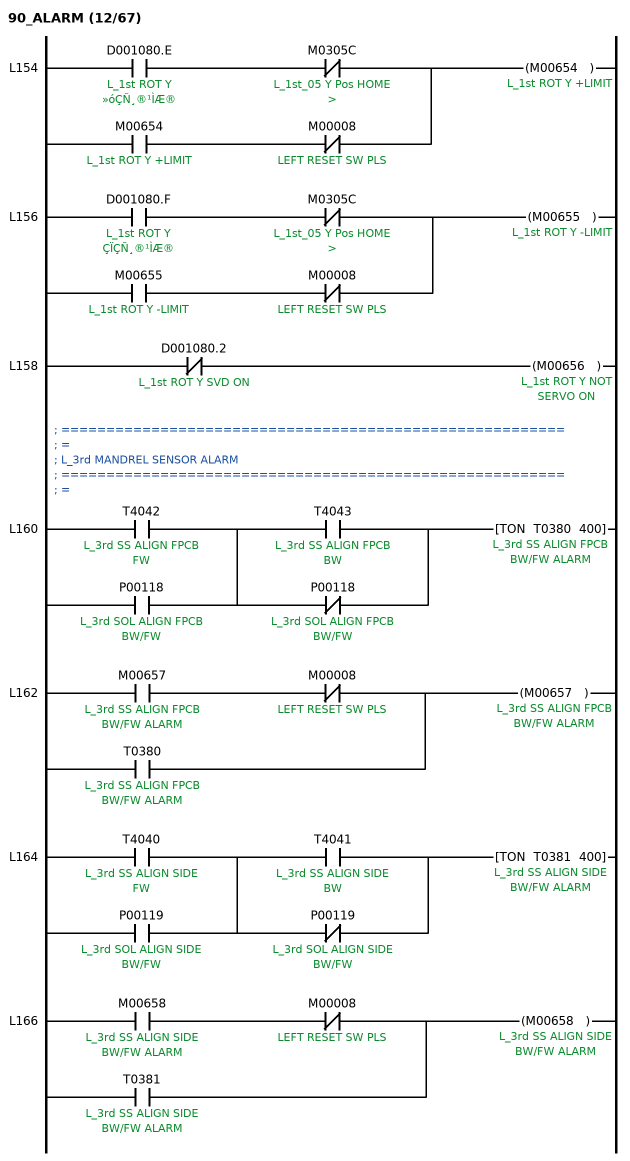
[picture p408: 90_ALARM rungs L154-L166]
; L154
LOAD      D001080.E	// L_1st ROT Y »óÇÑ¸®¹ÌÆ®
AND NOT   M0305C	// L_1st_05 Y Pos HOME >
LOAD      M00654	// L_1st ROT Y +LIMIT
AND NOT   M00008	// LEFT RESET SW PLS
OR LOAD
OUT       M00654	// L_1st ROT Y +LIMIT
; L156
LOAD      D001080.F	// L_1st ROT Y ÇÏÇÑ¸®¹ÌÆ®
AND NOT   M0305C	// L_1st_05 Y Pos HOME >
LOAD      M00655	// L_1st ROT Y -LIMIT
AND NOT   M00008	// LEFT RESET SW PLS
OR LOAD
OUT       M00655	// L_1st ROT Y -LIMIT
; L158
LOAD NOT  D001080.2	// L_1st ROT Y SVD ON
OUT       M00656	// L_1st ROT Y NOT SERVO ON
// =========================================================
// 
//        L_3rd MANDREL SENSOR ALARM
// 
// =========================================================
; L160
LOAD      T4042	// L_3rd SS ALIGN FPCB FW
OR        P00118	// L_3rd SOL ALIGN FPCB BW/FW
LOAD      T4043	// L_3rd SS ALIGN FPCB BW
OR NOT    P00118	// L_3rd SOL ALIGN FPCB BW/FW
AND LOAD
TON       T0380 400	// L_3rd SS ALIGN FPCB BW/FW ALARM
; L162
LOAD      M00657	// L_3rd SS ALIGN FPCB BW/FW ALARM
AND NOT   M00008	// LEFT RESET SW PLS
OR        T0380	// L_3rd SS ALIGN FPCB BW/FW ALARM
OUT       M00657	// L_3rd SS ALIGN FPCB BW/FW ALARM
; L164
LOAD      T4040	// L_3rd SS ALIGN SIDE FW
OR        P00119	// L_3rd SOL ALIGN SIDE BW/FW
LOAD      T4041	// L_3rd SS ALIGN SIDE BW
OR NOT    P00119	// L_3rd SOL ALIGN SIDE BW/FW
AND LOAD
TON       T0381 400	// L_3rd SS ALIGN SIDE BW/FW ALARM
; L166
LOAD      M00658	// L_3rd SS ALIGN SIDE BW/FW ALARM
AND NOT   M00008	// LEFT RESET SW PLS
OR        T0381	// L_3rd SS ALIGN SIDE BW/FW ALARM
OUT       M00658	// L_3rd SS ALIGN SIDE BW/FW ALARM

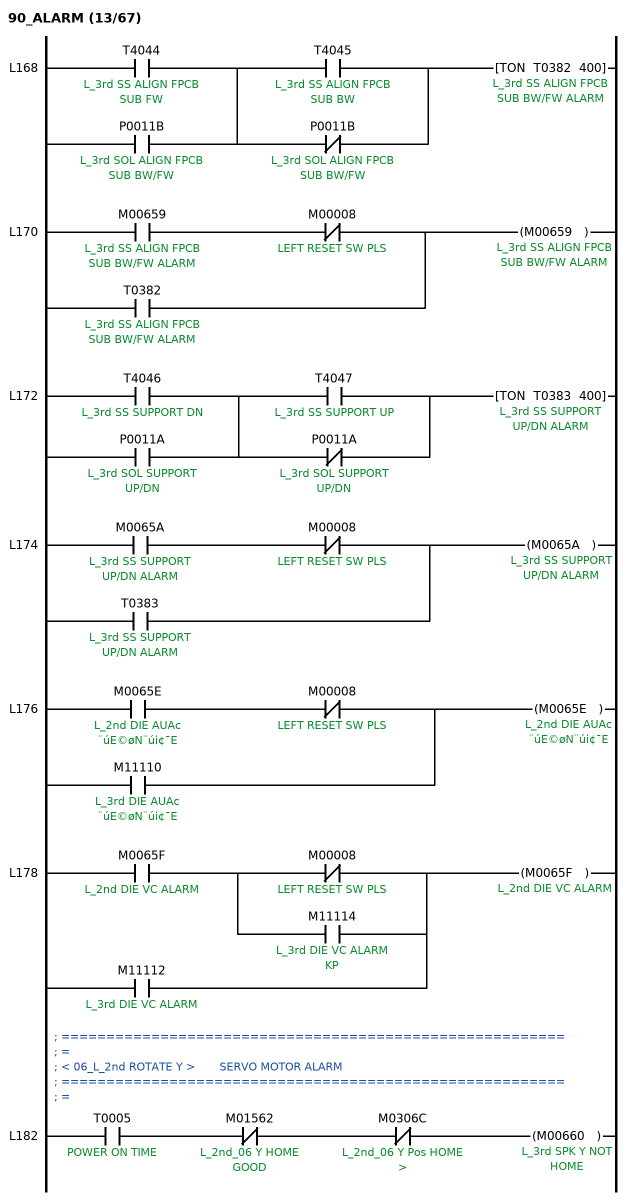
; L168
LOAD      T4044	// L_3rd SS ALIGN FPCB SUB FW
OR        P0011B	// L_3rd SOL ALIGN FPCB SUB BW/FW
LOAD      T4045	// L_3rd SS ALIGN FPCB SUB BW
OR NOT    P0011B	// L_3rd SOL ALIGN FPCB SUB BW/FW
AND LOAD
TON       T0382 400	// L_3rd SS ALIGN FPCB SUB BW/FW ALARM
; L170
LOAD      M00659	// L_3rd SS ALIGN FPCB SUB BW/FW ALARM
AND NOT   M00008	// LEFT RESET SW PLS
OR        T0382	// L_3rd SS ALIGN FPCB SUB BW/FW ALARM
OUT       M00659	// L_3rd SS ALIGN FPCB SUB BW/FW ALARM
; L172
LOAD      T4046	// L_3rd SS SUPPORT DN
OR        P0011A	// L_3rd SOL SUPPORT UP/DN
LOAD      T4047	// L_3rd SS SUPPORT UP
OR NOT    P0011A	// L_3rd SOL SUPPORT UP/DN
AND LOAD
TON       T0383 400	// L_3rd SS SUPPORT UP/DN ALARM
; L174
LOAD      M0065A	// L_3rd SS SUPPORT UP/DN ALARM
AND NOT   M00008	// LEFT RESET SW PLS
OR        T0383	// L_3rd SS SUPPORT UP/DN ALARM
OUT       M0065A	// L_3rd SS SUPPORT UP/DN ALARM
; L176
LOAD      M0065E	// L_2nd DIE AUAc ¨úE©øN¨úi¢¯E
AND NOT   M00008	// LEFT RESET SW PLS
OR        M11110	// L_3rd DIE AUAc ¨úE©øN¨úi¢¯E
OUT       M0065E	// L_2nd DIE AUAc ¨úE©øN¨úi¢¯E
; L178
LOAD      M0065F	// L_2nd DIE VC ALARM
LOAD NOT  M00008	// LEFT RESET SW PLS
OR        M11114	// L_3rd DIE VC ALARM KP
AND LOAD
OR        M11112	// L_3rd DIE VC ALARM
OUT       M0065F	// L_2nd DIE VC ALARM
// =========================================================
// 
//        < 06_L_2nd ROTATE Y >       SERVO MOTOR ALARM
// 
// =========================================================
; L182
LOAD      T0005	// POWER ON TIME
AND NOT   M01562	// L_2nd_06 Y HOME GOOD
AND NOT   M0306C	// L_2nd_06 Y Pos HOME >
OUT       M00660	// L_3rd SPK Y NOT HOME

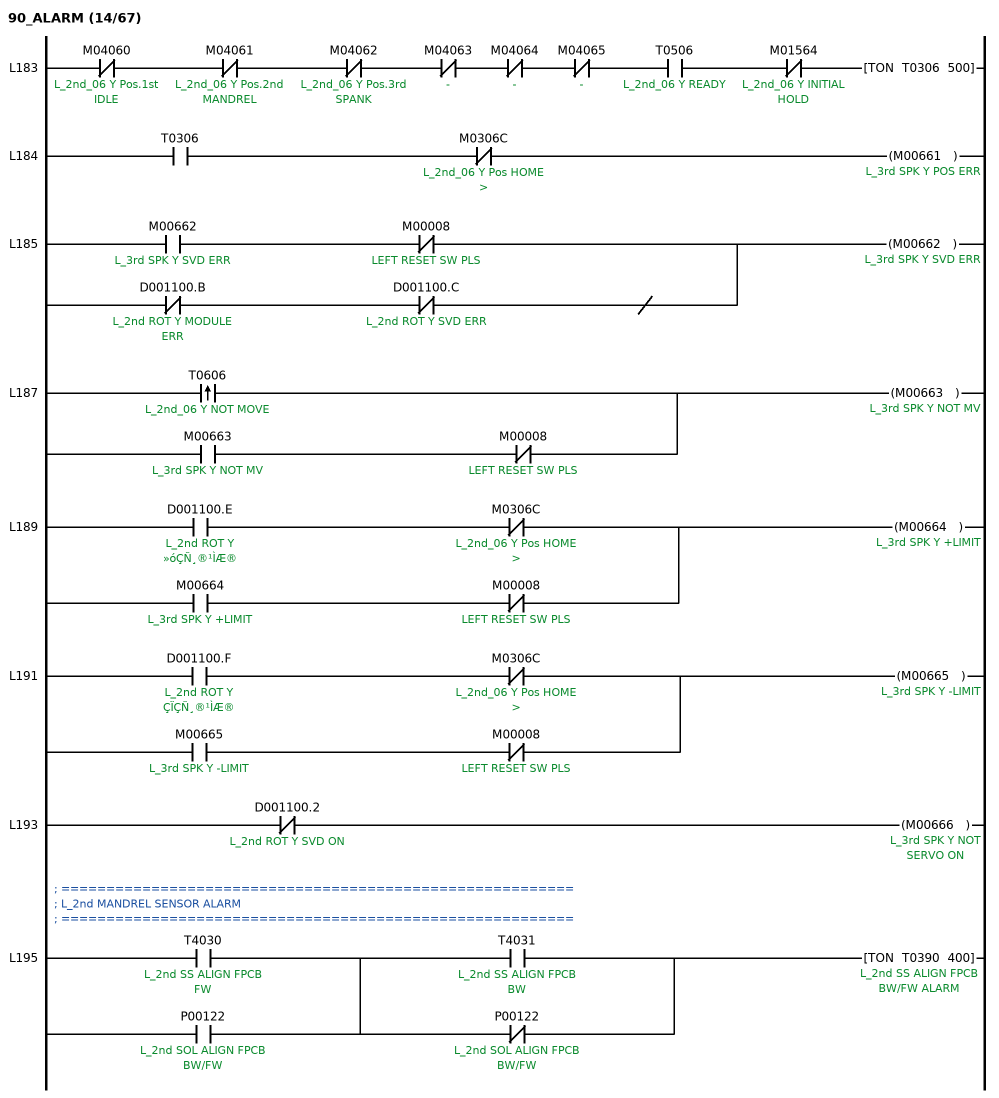
; L183
LOAD NOT  M04060	// L_2nd_06 Y Pos.1st IDLE
AND NOT   M04061	// L_2nd_06 Y Pos.2nd MANDREL
AND NOT   M04062	// L_2nd_06 Y Pos.3rd SPANK
AND NOT   M04063	// -
AND NOT   M04064	// -
AND NOT   M04065	// -
AND       T0506	// L_2nd_06 Y READY
AND NOT   M01564	// L_2nd_06 Y INITIAL HOLD
TON       T0306 500
; L184
LOAD      T0306
AND NOT   M0306C	// L_2nd_06 Y Pos HOME >
OUT       M00661	// L_3rd SPK Y POS ERR
; L185
LOAD      M00662	// L_3rd SPK Y SVD ERR
AND NOT   M00008	// LEFT RESET SW PLS
LOAD NOT  D001100.B	// L_2nd ROT Y MODULE ERR
AND NOT   D001100.C	// L_2nd ROT Y SVD ERR
NOT
OR LOAD
OUT       M00662	// L_3rd SPK Y SVD ERR
; L187
LOADP     T0606	// L_2nd_06 Y NOT MOVE
LOAD      M00663	// L_3rd SPK Y NOT MV
AND NOT   M00008	// LEFT RESET SW PLS
OR LOAD
OUT       M00663	// L_3rd SPK Y NOT MV
; L189
LOAD      D001100.E	// L_2nd ROT Y »óÇÑ¸®¹ÌÆ®
AND NOT   M0306C	// L_2nd_06 Y Pos HOME >
LOAD      M00664	// L_3rd SPK Y +LIMIT
AND NOT   M00008	// LEFT RESET SW PLS
OR LOAD
OUT       M00664	// L_3rd SPK Y +LIMIT
; L191
LOAD      D001100.F	// L_2nd ROT Y ÇÏÇÑ¸®¹ÌÆ®
AND NOT   M0306C	// L_2nd_06 Y Pos HOME >
LOAD      M00665	// L_3rd SPK Y -LIMIT
AND NOT   M00008	// LEFT RESET SW PLS
OR LOAD
OUT       M00665	// L_3rd SPK Y -LIMIT
; L193
LOAD NOT  D001100.2	// L_2nd ROT Y SVD ON
OUT       M00666	// L_3rd SPK Y NOT SERVO ON
// =========================================================
// 
//        L_2nd MANDREL SENSOR ALARM
// 
// =========================================================
; L195
LOAD      T4030	// L_2nd SS ALIGN FPCB FW
OR        P00122	// L_2nd SOL ALIGN FPCB BW/FW
LOAD      T4031	// L_2nd SS ALIGN FPCB BW
OR NOT    P00122	// L_2nd SOL ALIGN FPCB BW/FW
AND LOAD
TON       T0390 400	// L_2nd SS ALIGN FPCB BW/FW ALARM

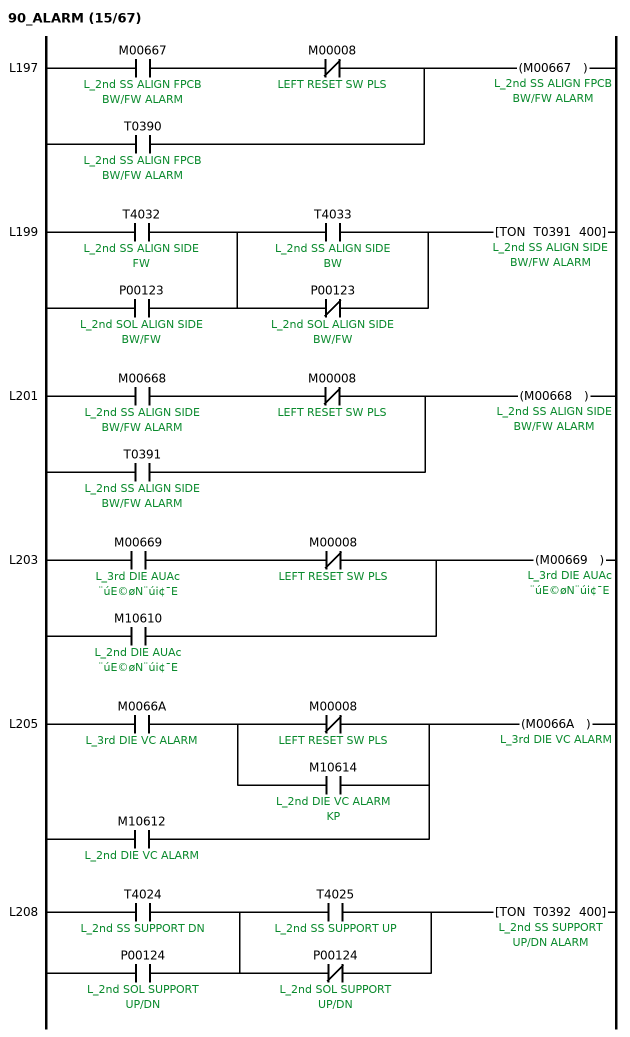
; L197
LOAD      M00667	// L_2nd SS ALIGN FPCB BW/FW ALARM
AND NOT   M00008	// LEFT RESET SW PLS
OR        T0390	// L_2nd SS ALIGN FPCB BW/FW ALARM
OUT       M00667	// L_2nd SS ALIGN FPCB BW/FW ALARM
; L199
LOAD      T4032	// L_2nd SS ALIGN SIDE FW
OR        P00123	// L_2nd SOL ALIGN SIDE BW/FW
LOAD      T4033	// L_2nd SS ALIGN SIDE BW
OR NOT    P00123	// L_2nd SOL ALIGN SIDE BW/FW
AND LOAD
TON       T0391 400	// L_2nd SS ALIGN SIDE BW/FW ALARM
; L201
LOAD      M00668	// L_2nd SS ALIGN SIDE BW/FW ALARM
AND NOT   M00008	// LEFT RESET SW PLS
OR        T0391	// L_2nd SS ALIGN SIDE BW/FW ALARM
OUT       M00668	// L_2nd SS ALIGN SIDE BW/FW ALARM
; L203
LOAD      M00669	// L_3rd DIE AUAc ¨úE©øN¨úi¢¯E
AND NOT   M00008	// LEFT RESET SW PLS
OR        M10610	// L_2nd DIE AUAc ¨úE©øN¨úi¢¯E
OUT       M00669	// L_3rd DIE AUAc ¨úE©øN¨úi¢¯E
; L205
LOAD      M0066A	// L_3rd DIE VC ALARM
LOAD NOT  M00008	// LEFT RESET SW PLS
OR        M10614	// L_2nd DIE VC ALARM KP
AND LOAD
OR        M10612	// L_2nd DIE VC ALARM
OUT       M0066A	// L_3rd DIE VC ALARM
; L208
LOAD      T4024	// L_2nd SS SUPPORT DN
OR        P00124	// L_2nd SOL SUPPORT UP/DN
LOAD      T4025	// L_2nd SS SUPPORT UP
OR NOT    P00124	// L_2nd SOL SUPPORT UP/DN
AND LOAD
TON       T0392 400	// L_2nd SS SUPPORT UP/DN ALARM

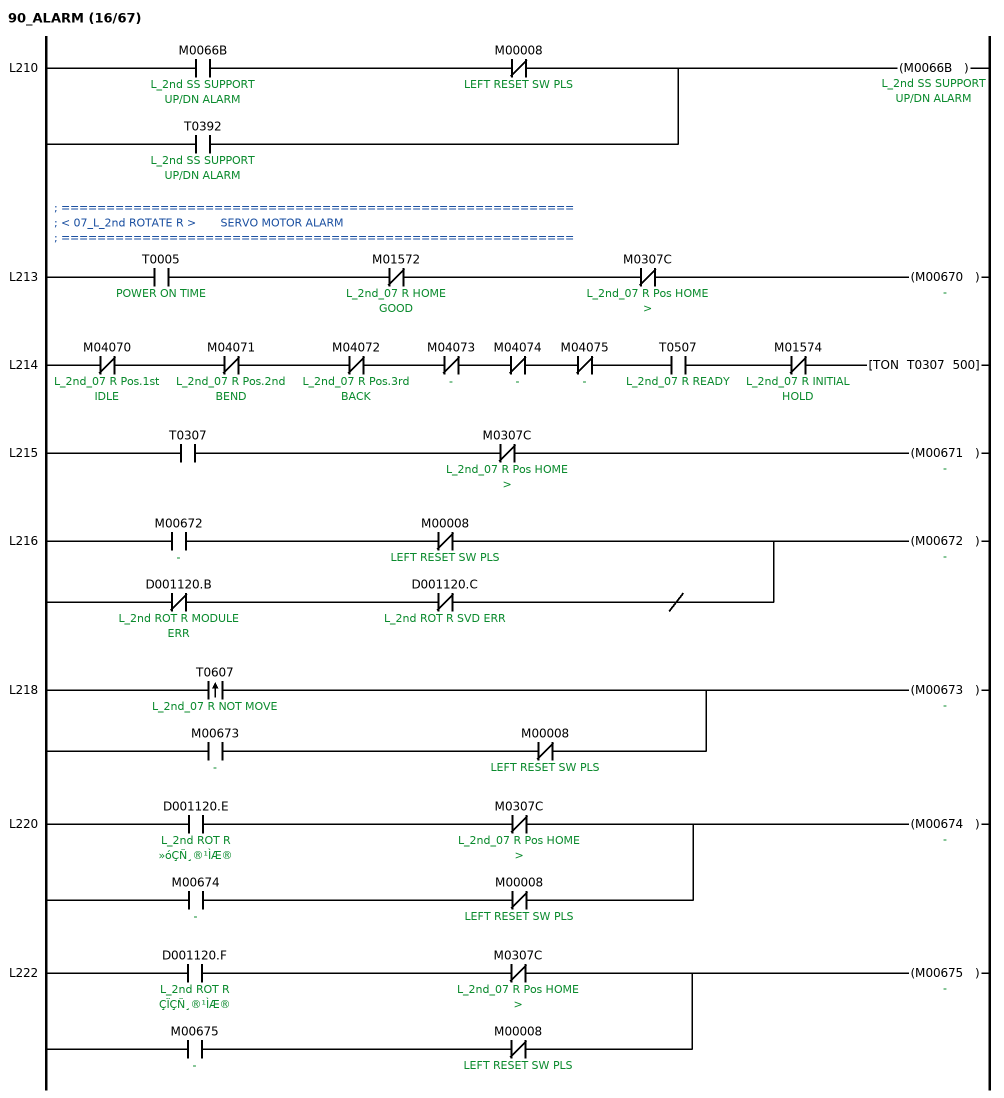
; L210
LOAD      M0066B	// L_2nd SS SUPPORT UP/DN ALARM
AND NOT   M00008	// LEFT RESET SW PLS
OR        T0392	// L_2nd SS SUPPORT UP/DN ALARM
OUT       M0066B	// L_2nd SS SUPPORT UP/DN ALARM
// =========================================================
// 
//        < 07_L_2nd ROTATE R >       SERVO MOTOR ALARM
// 
// =========================================================
; L213
LOAD      T0005	// POWER ON TIME
AND NOT   M01572	// L_2nd_07 R HOME GOOD
AND NOT   M0307C	// L_2nd_07 R Pos HOME >
OUT       M00670	// -
; L214
LOAD NOT  M04070	// L_2nd_07 R Pos.1st IDLE
AND NOT   M04071	// L_2nd_07 R Pos.2nd BEND
AND NOT   M04072	// L_2nd_07 R Pos.3rd BACK
AND NOT   M04073	// -
AND NOT   M04074	// -
AND NOT   M04075	// -
AND       T0507	// L_2nd_07 R READY
AND NOT   M01574	// L_2nd_07 R INITIAL HOLD
TON       T0307 500
; L215
LOAD      T0307
AND NOT   M0307C	// L_2nd_07 R Pos HOME >
OUT       M00671	// -
; L216
LOAD      M00672	// -
AND NOT   M00008	// LEFT RESET SW PLS
LOAD NOT  D001120.B	// L_2nd ROT R MODULE ERR
AND NOT   D001120.C	// L_2nd ROT R SVD ERR
NOT
OR LOAD
OUT       M00672	// -
; L218
LOADP     T0607	// L_2nd_07 R NOT MOVE
LOAD      M00673	// -
AND NOT   M00008	// LEFT RESET SW PLS
OR LOAD
OUT       M00673	// -
; L220
LOAD      D001120.E	// L_2nd ROT R »óÇÑ¸®¹ÌÆ®
AND NOT   M0307C	// L_2nd_07 R Pos HOME >
LOAD      M00674	// -
AND NOT   M00008	// LEFT RESET SW PLS
OR LOAD
OUT       M00674	// -
; L222
LOAD      D001120.F	// L_2nd ROT R ÇÏÇÑ¸®¹ÌÆ®
AND NOT   M0307C	// L_2nd_07 R Pos HOME >
LOAD      M00675	// -
AND NOT   M00008	// LEFT RESET SW PLS
OR LOAD
OUT       M00675	// -

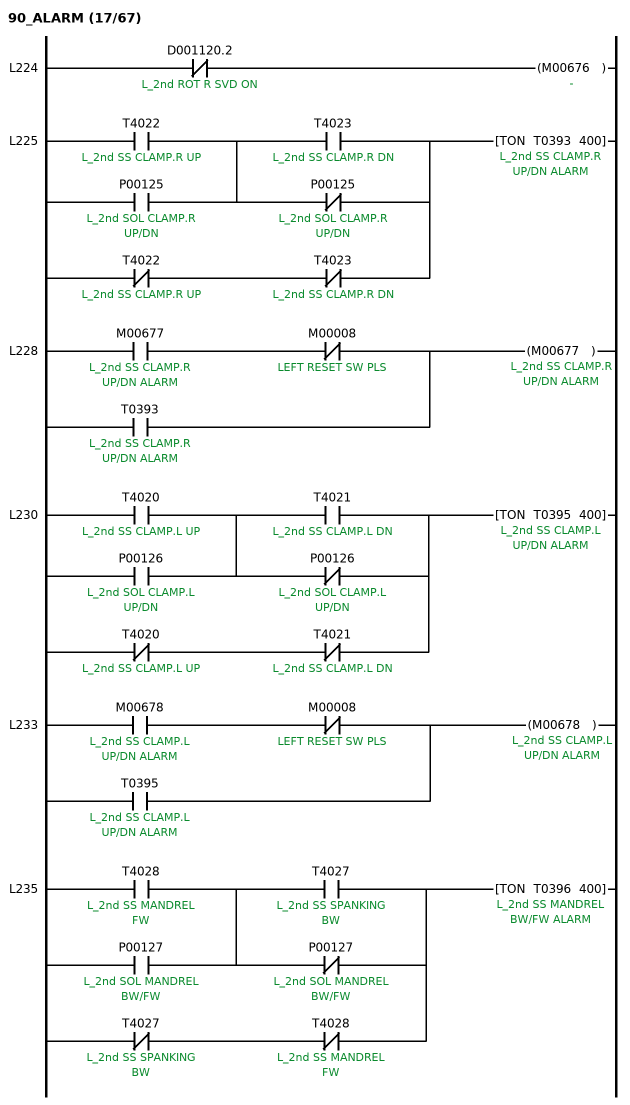
; L224
LOAD NOT  D001120.2	// L_2nd ROT R SVD ON
OUT       M00676	// -
; L225
LOAD      T4022	// L_2nd SS CLAMP.R UP
OR        P00125	// L_2nd SOL CLAMP.R UP/DN
LOAD      T4023	// L_2nd SS CLAMP.R DN
OR NOT    P00125	// L_2nd SOL CLAMP.R UP/DN
AND LOAD
LOAD NOT  T4022	// L_2nd SS CLAMP.R UP
AND NOT   T4023	// L_2nd SS CLAMP.R DN
OR LOAD
TON       T0393 400	// L_2nd SS CLAMP.R UP/DN ALARM
; L228
LOAD      M00677	// L_2nd SS CLAMP.R UP/DN ALARM
AND NOT   M00008	// LEFT RESET SW PLS
OR        T0393	// L_2nd SS CLAMP.R UP/DN ALARM
OUT       M00677	// L_2nd SS CLAMP.R UP/DN ALARM
; L230
LOAD      T4020	// L_2nd SS CLAMP.L UP
OR        P00126	// L_2nd SOL CLAMP.L UP/DN
LOAD      T4021	// L_2nd SS CLAMP.L DN
OR NOT    P00126	// L_2nd SOL CLAMP.L UP/DN
AND LOAD
LOAD NOT  T4020	// L_2nd SS CLAMP.L UP
AND NOT   T4021	// L_2nd SS CLAMP.L DN
OR LOAD
TON       T0395 400	// L_2nd SS CLAMP.L UP/DN ALARM
; L233
LOAD      M00678	// L_2nd SS CLAMP.L UP/DN ALARM
AND NOT   M00008	// LEFT RESET SW PLS
OR        T0395	// L_2nd SS CLAMP.L UP/DN ALARM
OUT       M00678	// L_2nd SS CLAMP.L UP/DN ALARM
; L235
LOAD      T4028	// L_2nd SS MANDREL FW
OR        P00127	// L_2nd SOL MANDREL BW/FW
LOAD      T4027	// L_2nd SS SPANKING BW
OR NOT    P00127	// L_2nd SOL MANDREL BW/FW
AND LOAD
LOAD NOT  T4027	// L_2nd SS SPANKING BW
AND NOT   T4028	// L_2nd SS MANDREL FW
OR LOAD
TON       T0396 400	// L_2nd SS MANDREL BW/FW ALARM

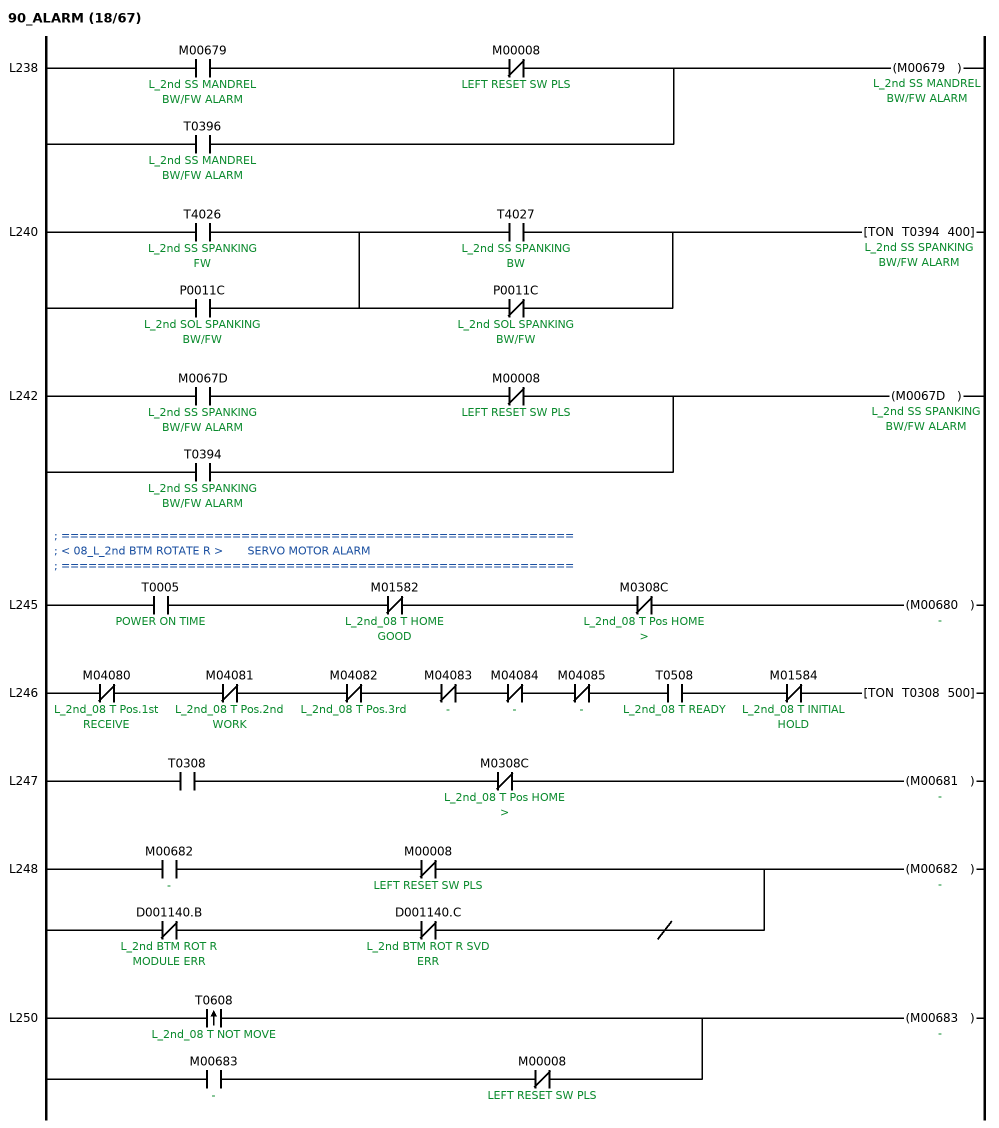
; L238
LOAD      M00679	// L_2nd SS MANDREL BW/FW ALARM
AND NOT   M00008	// LEFT RESET SW PLS
OR        T0396	// L_2nd SS MANDREL BW/FW ALARM
OUT       M00679	// L_2nd SS MANDREL BW/FW ALARM
; L240
LOAD      T4026	// L_2nd SS SPANKING FW
OR        P0011C	// L_2nd SOL SPANKING BW/FW
LOAD      T4027	// L_2nd SS SPANKING BW
OR NOT    P0011C	// L_2nd SOL SPANKING BW/FW
AND LOAD
TON       T0394 400	// L_2nd SS SPANKING BW/FW ALARM
; L242
LOAD      M0067D	// L_2nd SS SPANKING BW/FW ALARM
AND NOT   M00008	// LEFT RESET SW PLS
OR        T0394	// L_2nd SS SPANKING BW/FW ALARM
OUT       M0067D	// L_2nd SS SPANKING BW/FW ALARM
// =========================================================
// 
//        < 08_L_2nd BTM ROTATE R >       SERVO MOTOR ALARM
// 
// =========================================================
; L245
LOAD      T0005	// POWER ON TIME
AND NOT   M01582	// L_2nd_08 T HOME GOOD
AND NOT   M0308C	// L_2nd_08 T Pos HOME >
OUT       M00680	// -
; L246
LOAD NOT  M04080	// L_2nd_08 T Pos.1st RECEIVE
AND NOT   M04081	// L_2nd_08 T Pos.2nd WORK
AND NOT   M04082	// L_2nd_08 T Pos.3rd
AND NOT   M04083	// -
AND NOT   M04084	// -
AND NOT   M04085	// -
AND       T0508	// L_2nd_08 T READY
AND NOT   M01584	// L_2nd_08 T INITIAL HOLD
TON       T0308 500
; L247
LOAD      T0308
AND NOT   M0308C	// L_2nd_08 T Pos HOME >
OUT       M00681	// -
; L248
LOAD      M00682	// -
AND NOT   M00008	// LEFT RESET SW PLS
LOAD NOT  D001140.B	// L_2nd BTM ROT R MODULE ERR
AND NOT   D001140.C	// L_2nd BTM ROT R SVD ERR
NOT
OR LOAD
OUT       M00682	// -
; L250
LOADP     T0608	// L_2nd_08 T NOT MOVE
LOAD      M00683	// -
AND NOT   M00008	// LEFT RESET SW PLS
OR LOAD
OUT       M00683	// -

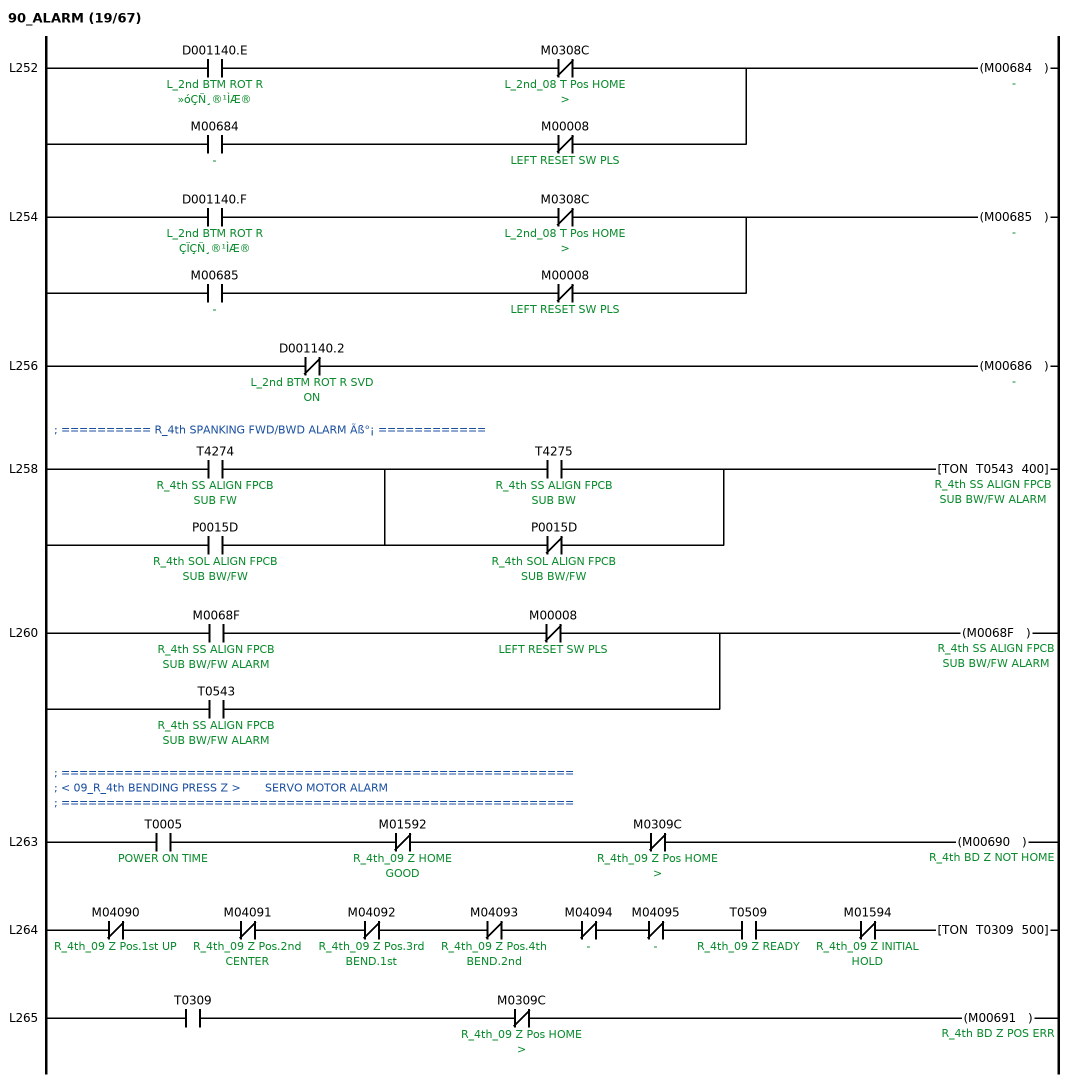
; L252
LOAD      D001140.E	// L_2nd BTM ROT R »óÇÑ¸®¹ÌÆ®
AND NOT   M0308C	// L_2nd_08 T Pos HOME >
LOAD      M00684	// -
AND NOT   M00008	// LEFT RESET SW PLS
OR LOAD
OUT       M00684	// -
; L254
LOAD      D001140.F	// L_2nd BTM ROT R ÇÏÇÑ¸®¹ÌÆ®
AND NOT   M0308C	// L_2nd_08 T Pos HOME >
LOAD      M00685	// -
AND NOT   M00008	// LEFT RESET SW PLS
OR LOAD
OUT       M00685	// -
; L256
LOAD NOT  D001140.2	// L_2nd BTM ROT R SVD ON
OUT       M00686	// -
// ========== R_4th SPANKING FWD/BWD ALARM Ãß°¡ ============
; L258
LOAD      T4274	// R_4th SS ALIGN FPCB SUB FW
OR        P0015D	// R_4th SOL ALIGN FPCB SUB BW/FW
LOAD      T4275	// R_4th SS ALIGN FPCB SUB BW
OR NOT    P0015D	// R_4th SOL ALIGN FPCB SUB BW/FW
AND LOAD
TON       T0543 400	// R_4th SS ALIGN FPCB SUB BW/FW ALARM
; L260
LOAD      M0068F	// R_4th SS ALIGN FPCB SUB BW/FW ALARM
AND NOT   M00008	// LEFT RESET SW PLS
OR        T0543	// R_4th SS ALIGN FPCB SUB BW/FW ALARM
OUT       M0068F	// R_4th SS ALIGN FPCB SUB BW/FW ALARM
// =========================================================
// 
//        < 09_R_4th BENDING PRESS Z >       SERVO MOTOR ALARM
// 
// =========================================================
; L263
LOAD      T0005	// POWER ON TIME
AND NOT   M01592	// R_4th_09 Z HOME GOOD
AND NOT   M0309C	// R_4th_09 Z Pos HOME >
OUT       M00690	// R_4th BD Z NOT HOME
; L264
LOAD NOT  M04090	// R_4th_09 Z Pos.1st UP
AND NOT   M04091	// R_4th_09 Z Pos.2nd CENTER
AND NOT   M04092	// R_4th_09 Z Pos.3rd BEND.1st
AND NOT   M04093	// R_4th_09 Z Pos.4th BEND.2nd
AND NOT   M04094	// -
AND NOT   M04095	// -
AND       T0509	// R_4th_09 Z READY
AND NOT   M01594	// R_4th_09 Z INITIAL HOLD
TON       T0309 500
; L265
LOAD      T0309
AND NOT   M0309C	// R_4th_09 Z Pos HOME >
OUT       M00691	// R_4th BD Z POS ERR

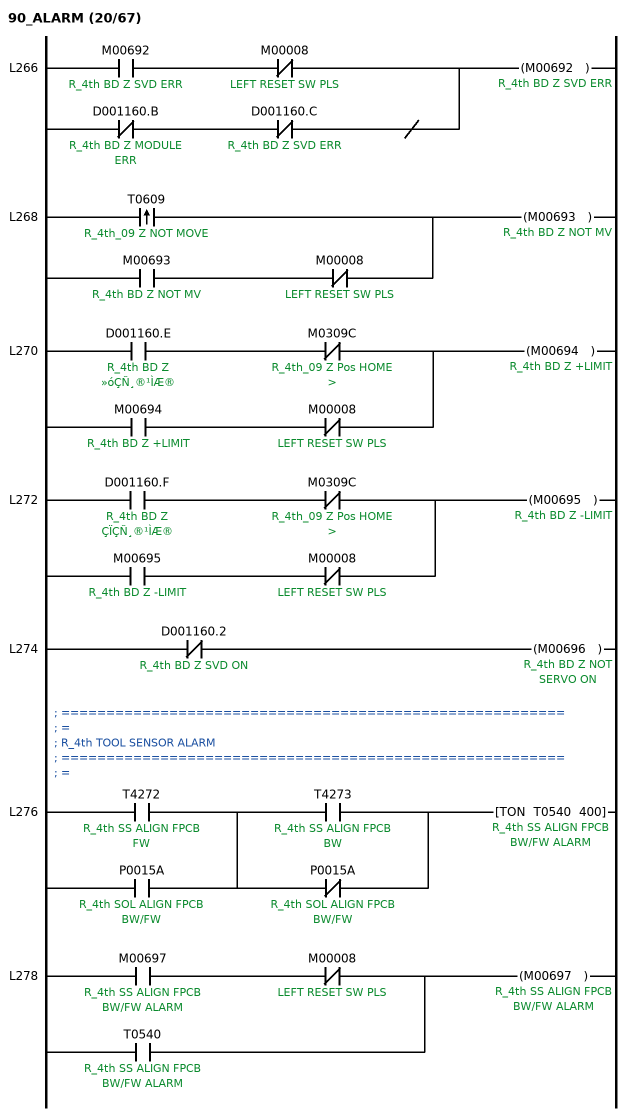
; L266
LOAD      M00692	// R_4th BD Z SVD ERR
AND NOT   M00008	// LEFT RESET SW PLS
LOAD NOT  D001160.B	// R_4th BD Z MODULE ERR
AND NOT   D001160.C	// R_4th BD Z SVD ERR
NOT
OR LOAD
OUT       M00692	// R_4th BD Z SVD ERR
; L268
LOADP     T0609	// R_4th_09 Z NOT MOVE
LOAD      M00693	// R_4th BD Z NOT MV
AND NOT   M00008	// LEFT RESET SW PLS
OR LOAD
OUT       M00693	// R_4th BD Z NOT MV
; L270
LOAD      D001160.E	// R_4th BD Z »óÇÑ¸®¹ÌÆ®
AND NOT   M0309C	// R_4th_09 Z Pos HOME >
LOAD      M00694	// R_4th BD Z +LIMIT
AND NOT   M00008	// LEFT RESET SW PLS
OR LOAD
OUT       M00694	// R_4th BD Z +LIMIT
; L272
LOAD      D001160.F	// R_4th BD Z ÇÏÇÑ¸®¹ÌÆ®
AND NOT   M0309C	// R_4th_09 Z Pos HOME >
LOAD      M00695	// R_4th BD Z -LIMIT
AND NOT   M00008	// LEFT RESET SW PLS
OR LOAD
OUT       M00695	// R_4th BD Z -LIMIT
; L274
LOAD NOT  D001160.2	// R_4th BD Z SVD ON
OUT       M00696	// R_4th BD Z NOT SERVO ON
// =========================================================
// 
//        R_4th TOOL SENSOR ALARM
// 
// =========================================================
; L276
LOAD      T4272	// R_4th SS ALIGN FPCB FW
OR        P0015A	// R_4th SOL ALIGN FPCB BW/FW
LOAD      T4273	// R_4th SS ALIGN FPCB BW
OR NOT    P0015A	// R_4th SOL ALIGN FPCB BW/FW
AND LOAD
TON       T0540 400	// R_4th SS ALIGN FPCB BW/FW ALARM
; L278
LOAD      M00697	// R_4th SS ALIGN FPCB BW/FW ALARM
AND NOT   M00008	// LEFT RESET SW PLS
OR        T0540	// R_4th SS ALIGN FPCB BW/FW ALARM
OUT       M00697	// R_4th SS ALIGN FPCB BW/FW ALARM

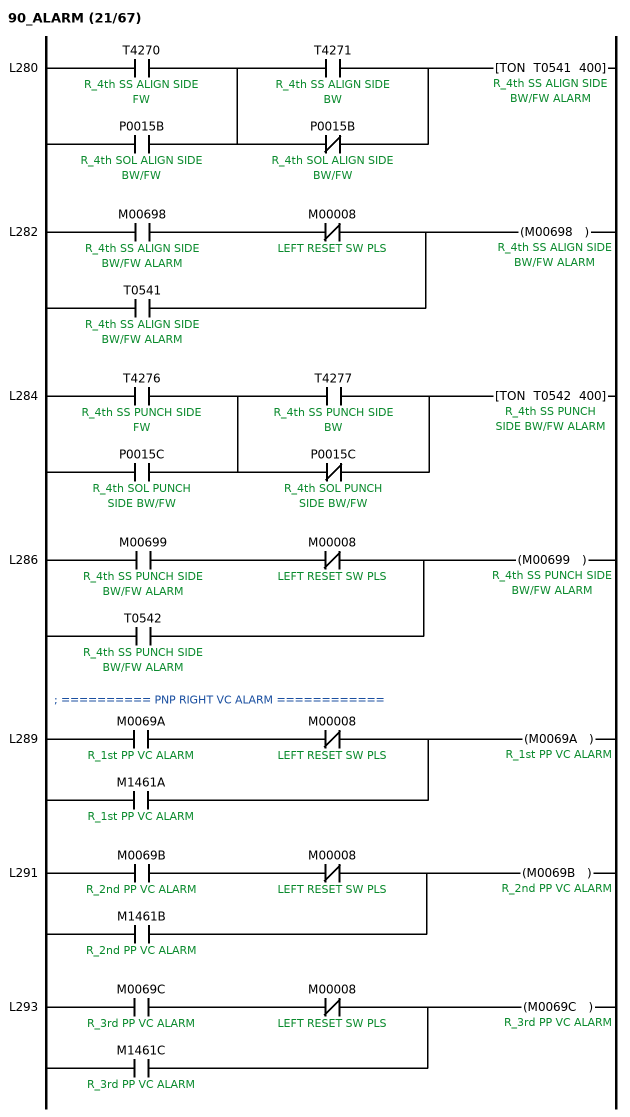
; L280
LOAD      T4270	// R_4th SS ALIGN SIDE FW
OR        P0015B	// R_4th SOL ALIGN SIDE BW/FW
LOAD      T4271	// R_4th SS ALIGN SIDE BW
OR NOT    P0015B	// R_4th SOL ALIGN SIDE BW/FW
AND LOAD
TON       T0541 400	// R_4th SS ALIGN SIDE BW/FW ALARM
; L282
LOAD      M00698	// R_4th SS ALIGN SIDE BW/FW ALARM
AND NOT   M00008	// LEFT RESET SW PLS
OR        T0541	// R_4th SS ALIGN SIDE BW/FW ALARM
OUT       M00698	// R_4th SS ALIGN SIDE BW/FW ALARM
; L284
LOAD      T4276	// R_4th SS PUNCH SIDE FW
OR        P0015C	// R_4th SOL PUNCH SIDE BW/FW
LOAD      T4277	// R_4th SS PUNCH SIDE BW
OR NOT    P0015C	// R_4th SOL PUNCH SIDE BW/FW
AND LOAD
TON       T0542 400	// R_4th SS PUNCH SIDE BW/FW ALARM
; L286
LOAD      M00699	// R_4th SS PUNCH SIDE BW/FW ALARM
AND NOT   M00008	// LEFT RESET SW PLS
OR        T0542	// R_4th SS PUNCH SIDE BW/FW ALARM
OUT       M00699	// R_4th SS PUNCH SIDE BW/FW ALARM
// ========== PNP RIGHT VC ALARM ============
; L289
LOAD      M0069A	// R_1st PP VC ALARM
AND NOT   M00008	// LEFT RESET SW PLS
OR        M1461A	// R_1st PP VC ALARM
OUT       M0069A	// R_1st PP VC ALARM
; L291
LOAD      M0069B	// R_2nd PP VC ALARM
AND NOT   M00008	// LEFT RESET SW PLS
OR        M1461B	// R_2nd PP VC ALARM
OUT       M0069B	// R_2nd PP VC ALARM
; L293
LOAD      M0069C	// R_3rd PP VC ALARM
AND NOT   M00008	// LEFT RESET SW PLS
OR        M1461C	// R_3rd PP VC ALARM
OUT       M0069C	// R_3rd PP VC ALARM

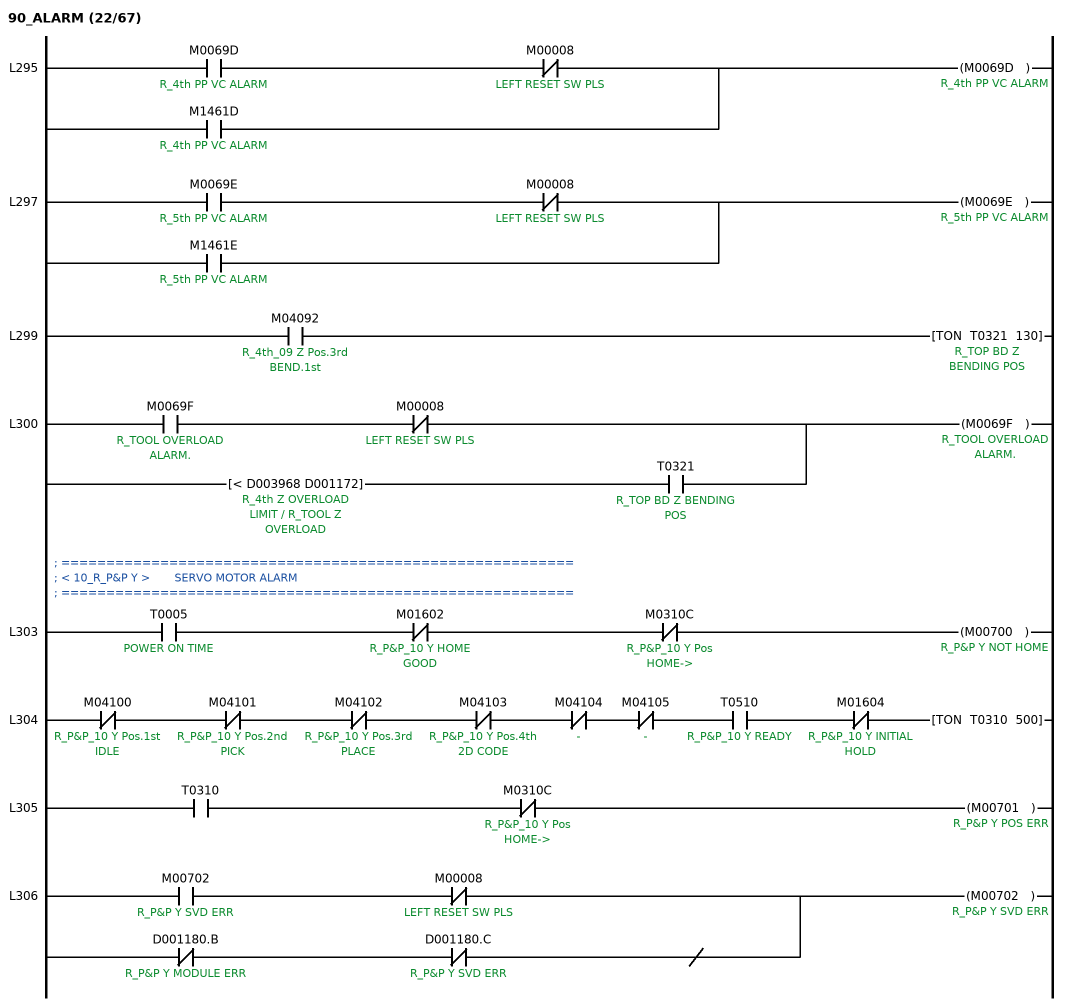
; L295
LOAD      M0069D	// R_4th PP VC ALARM
AND NOT   M00008	// LEFT RESET SW PLS
OR        M1461D	// R_4th PP VC ALARM
OUT       M0069D	// R_4th PP VC ALARM
; L297
LOAD      M0069E	// R_5th PP VC ALARM
AND NOT   M00008	// LEFT RESET SW PLS
OR        M1461E	// R_5th PP VC ALARM
OUT       M0069E	// R_5th PP VC ALARM
; L299
LOAD      M04092	// R_4th_09 Z Pos.3rd BEND.1st
TON       T0321 130	// R_TOP BD Z BENDING POS
; L300
LOAD      M0069F	// R_TOOL OVERLOAD ALARM.
AND NOT   M00008	// LEFT RESET SW PLS
LOAD<     D003968 D001172	// R_4th Z OVERLOAD LIMIT / R_TOOL Z OVERLOAD
AND       T0321	// R_TOP BD Z BENDING POS
OR LOAD
OUT       M0069F	// R_TOOL OVERLOAD ALARM.
// =========================================================
// 
//        < 10_R_P&P Y >       SERVO MOTOR ALARM
// 
// =========================================================
; L303
LOAD      T0005	// POWER ON TIME
AND NOT   M01602	// R_P&P_10 Y HOME GOOD
AND NOT   M0310C	// R_P&P_10 Y Pos HOME->
OUT       M00700	// R_P&P Y NOT HOME
; L304
LOAD NOT  M04100	// R_P&P_10 Y Pos.1st IDLE
AND NOT   M04101	// R_P&P_10 Y Pos.2nd PICK
AND NOT   M04102	// R_P&P_10 Y Pos.3rd PLACE
AND NOT   M04103	// R_P&P_10 Y Pos.4th 2D CODE
AND NOT   M04104	// -
AND NOT   M04105	// -
AND       T0510	// R_P&P_10 Y READY
AND NOT   M01604	// R_P&P_10 Y INITIAL HOLD
TON       T0310 500
; L305
LOAD      T0310
AND NOT   M0310C	// R_P&P_10 Y Pos HOME->
OUT       M00701	// R_P&P Y POS ERR
; L306
LOAD      M00702	// R_P&P Y SVD ERR
AND NOT   M00008	// LEFT RESET SW PLS
LOAD NOT  D001180.B	// R_P&P Y MODULE ERR
AND NOT   D001180.C	// R_P&P Y SVD ERR
NOT
OR LOAD
OUT       M00702	// R_P&P Y SVD ERR

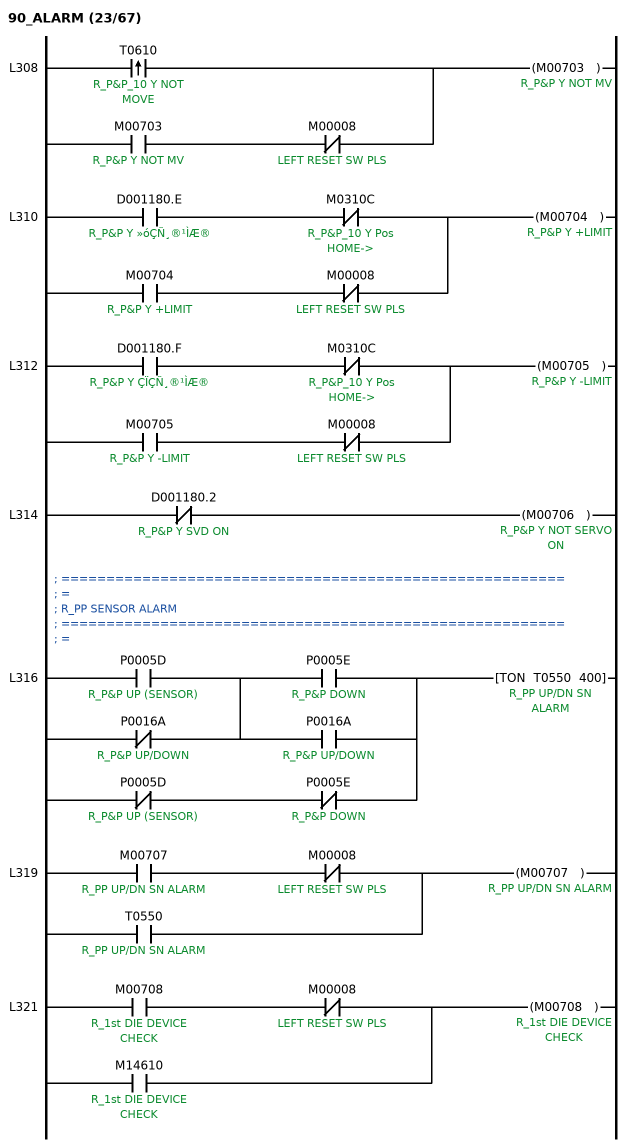
; L308
LOADP     T0610	// R_P&P_10 Y NOT MOVE
LOAD      M00703	// R_P&P Y NOT MV
AND NOT   M00008	// LEFT RESET SW PLS
OR LOAD
OUT       M00703	// R_P&P Y NOT MV
; L310
LOAD      D001180.E	// R_P&P Y »óÇÑ¸®¹ÌÆ®
AND NOT   M0310C	// R_P&P_10 Y Pos HOME->
LOAD      M00704	// R_P&P Y +LIMIT
AND NOT   M00008	// LEFT RESET SW PLS
OR LOAD
OUT       M00704	// R_P&P Y +LIMIT
; L312
LOAD      D001180.F	// R_P&P Y ÇÏÇÑ¸®¹ÌÆ®
AND NOT   M0310C	// R_P&P_10 Y Pos HOME->
LOAD      M00705	// R_P&P Y -LIMIT
AND NOT   M00008	// LEFT RESET SW PLS
OR LOAD
OUT       M00705	// R_P&P Y -LIMIT
; L314
LOAD NOT  D001180.2	// R_P&P Y SVD ON
OUT       M00706	// R_P&P Y NOT SERVO ON
// =========================================================
// 
//       R_PP SENSOR ALARM
// 
// =========================================================
; L316
LOAD      P0005D	// R_P&P UP (SENSOR)
OR NOT    P0016A	// R_P&P UP/DOWN
LOAD      P0005E	// R_P&P DOWN
OR        P0016A	// R_P&P UP/DOWN
AND LOAD
LOAD NOT  P0005D	// R_P&P UP (SENSOR)
AND NOT   P0005E	// R_P&P DOWN
OR LOAD
TON       T0550 400	// R_PP UP/DN SN ALARM
; L319
LOAD      M00707	// R_PP UP/DN SN ALARM
AND NOT   M00008	// LEFT RESET SW PLS
OR        T0550	// R_PP UP/DN SN ALARM
OUT       M00707	// R_PP UP/DN SN ALARM
; L321
LOAD      M00708	// R_1st DIE DEVICE CHECK
AND NOT   M00008	// LEFT RESET SW PLS
OR        M14610	// R_1st DIE DEVICE CHECK
OUT       M00708	// R_1st DIE DEVICE CHECK

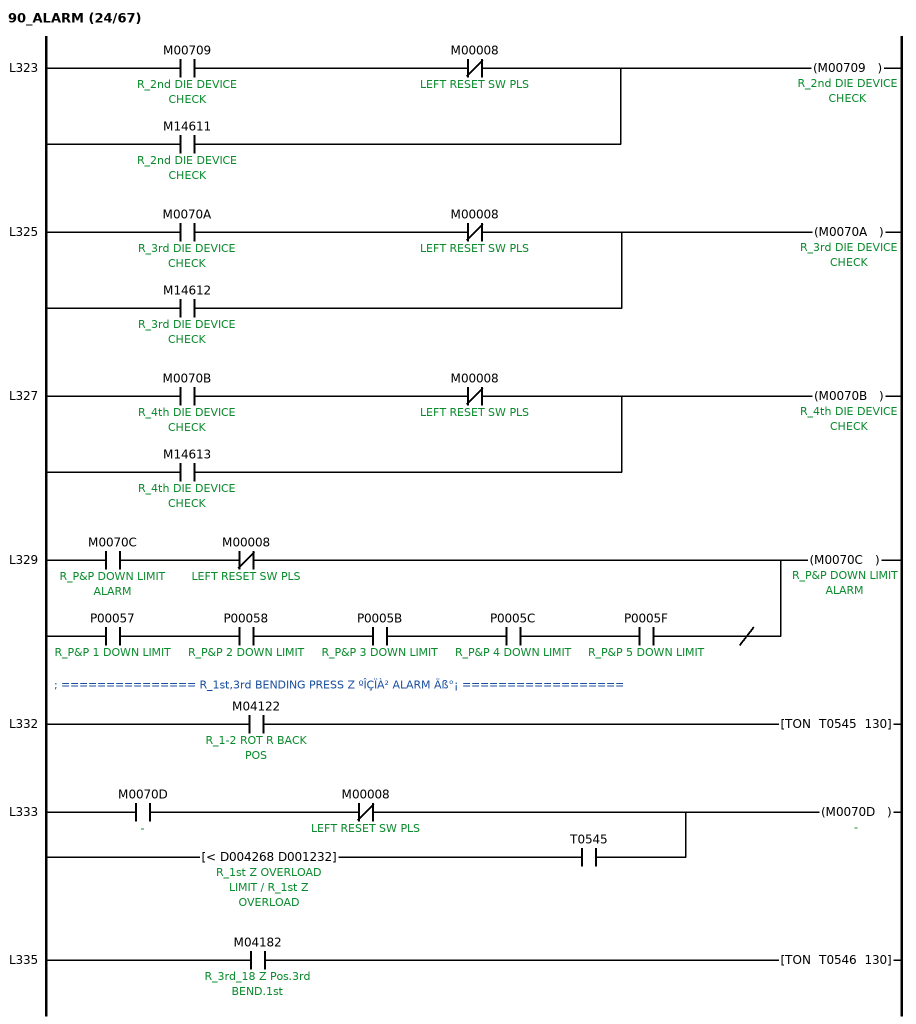
; L323
LOAD      M00709	// R_2nd DIE DEVICE CHECK
AND NOT   M00008	// LEFT RESET SW PLS
OR        M14611	// R_2nd DIE DEVICE CHECK
OUT       M00709	// R_2nd DIE DEVICE CHECK
; L325
LOAD      M0070A	// R_3rd DIE DEVICE CHECK
AND NOT   M00008	// LEFT RESET SW PLS
OR        M14612	// R_3rd DIE DEVICE CHECK
OUT       M0070A	// R_3rd DIE DEVICE CHECK
; L327
LOAD      M0070B	// R_4th DIE DEVICE CHECK
AND NOT   M00008	// LEFT RESET SW PLS
OR        M14613	// R_4th DIE DEVICE CHECK
OUT       M0070B	// R_4th DIE DEVICE CHECK
; L329
LOAD      M0070C	// R_P&P DOWN LIMIT ALARM
AND NOT   M00008	// LEFT RESET SW PLS
LOAD      P00057	// R_P&P 1 DOWN LIMIT
AND       P00058	// R_P&P 2 DOWN LIMIT
AND       P0005B	// R_P&P 3 DOWN LIMIT
AND       P0005C	// R_P&P 4 DOWN LIMIT
AND       P0005F	// R_P&P 5 DOWN LIMIT
NOT
OR LOAD
OUT       M0070C	// R_P&P DOWN LIMIT ALARM
// =============== R_1st,3rd BENDING PRESS Z ºÎÇÏÀ² ALARM Ãß°¡ ==================
; L332
LOAD      M04122	// R_1-2 ROT R BACK POS
TON       T0545 130
; L333
LOAD      M0070D	// -
AND NOT   M00008	// LEFT RESET SW PLS
LOAD<     D004268 D001232	// R_1st Z OVERLOAD LIMIT / R_1st Z OVERLOAD
AND       T0545
OR LOAD
OUT       M0070D	// -
; L335
LOAD      M04182	// R_3rd_18 Z Pos.3rd BEND.1st
TON       T0546 130

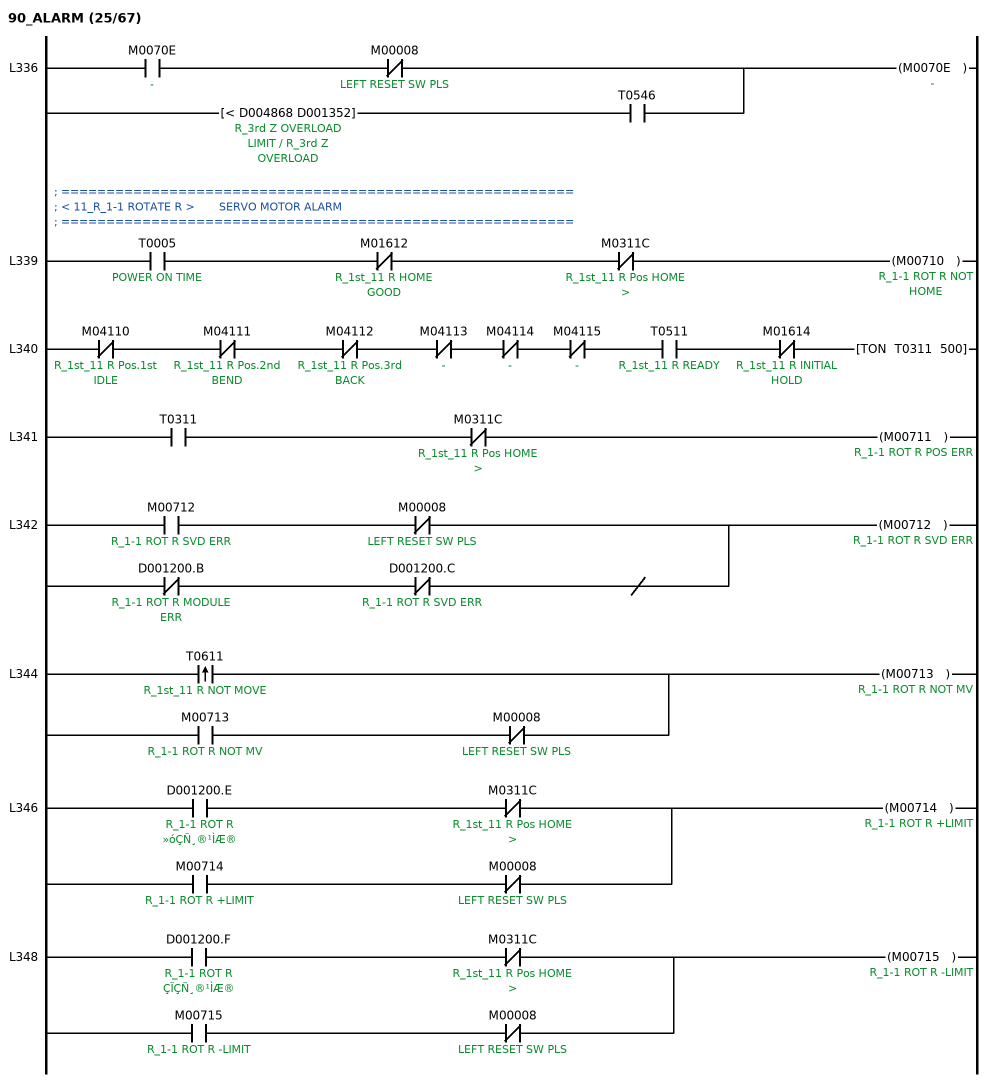
; L336
LOAD      M0070E	// -
AND NOT   M00008	// LEFT RESET SW PLS
LOAD<     D004868 D001352	// R_3rd Z OVERLOAD LIMIT / R_3rd Z OVERLOAD
AND       T0546
OR LOAD
OUT       M0070E	// -
// =========================================================
// 
//        < 11_R_1-1 ROTATE R >       SERVO MOTOR ALARM
// 
// =========================================================
; L339
LOAD      T0005	// POWER ON TIME
AND NOT   M01612	// R_1st_11 R HOME GOOD
AND NOT   M0311C	// R_1st_11 R Pos HOME >
OUT       M00710	// R_1-1 ROT R NOT HOME
; L340
LOAD NOT  M04110	// R_1st_11 R Pos.1st IDLE
AND NOT   M04111	// R_1st_11 R Pos.2nd BEND
AND NOT   M04112	// R_1st_11 R Pos.3rd BACK
AND NOT   M04113	// -
AND NOT   M04114	// -
AND NOT   M04115	// -
AND       T0511	// R_1st_11 R READY
AND NOT   M01614	// R_1st_11 R INITIAL HOLD
TON       T0311 500
; L341
LOAD      T0311
AND NOT   M0311C	// R_1st_11 R Pos HOME >
OUT       M00711	// R_1-1 ROT R POS ERR
; L342
LOAD      M00712	// R_1-1 ROT R SVD ERR
AND NOT   M00008	// LEFT RESET SW PLS
LOAD NOT  D001200.B	// R_1-1 ROT R MODULE ERR
AND NOT   D001200.C	// R_1-1 ROT R SVD ERR
NOT
OR LOAD
OUT       M00712	// R_1-1 ROT R SVD ERR
; L344
LOADP     T0611	// R_1st_11 R NOT MOVE
LOAD      M00713	// R_1-1 ROT R NOT MV
AND NOT   M00008	// LEFT RESET SW PLS
OR LOAD
OUT       M00713	// R_1-1 ROT R NOT MV
; L346
LOAD      D001200.E	// R_1-1 ROT R »óÇÑ¸®¹ÌÆ®
AND NOT   M0311C	// R_1st_11 R Pos HOME >
LOAD      M00714	// R_1-1 ROT R +LIMIT
AND NOT   M00008	// LEFT RESET SW PLS
OR LOAD
OUT       M00714	// R_1-1 ROT R +LIMIT
; L348
LOAD      D001200.F	// R_1-1 ROT R ÇÏÇÑ¸®¹ÌÆ®
AND NOT   M0311C	// R_1st_11 R Pos HOME >
LOAD      M00715	// R_1-1 ROT R -LIMIT
AND NOT   M00008	// LEFT RESET SW PLS
OR LOAD
OUT       M00715	// R_1-1 ROT R -LIMIT

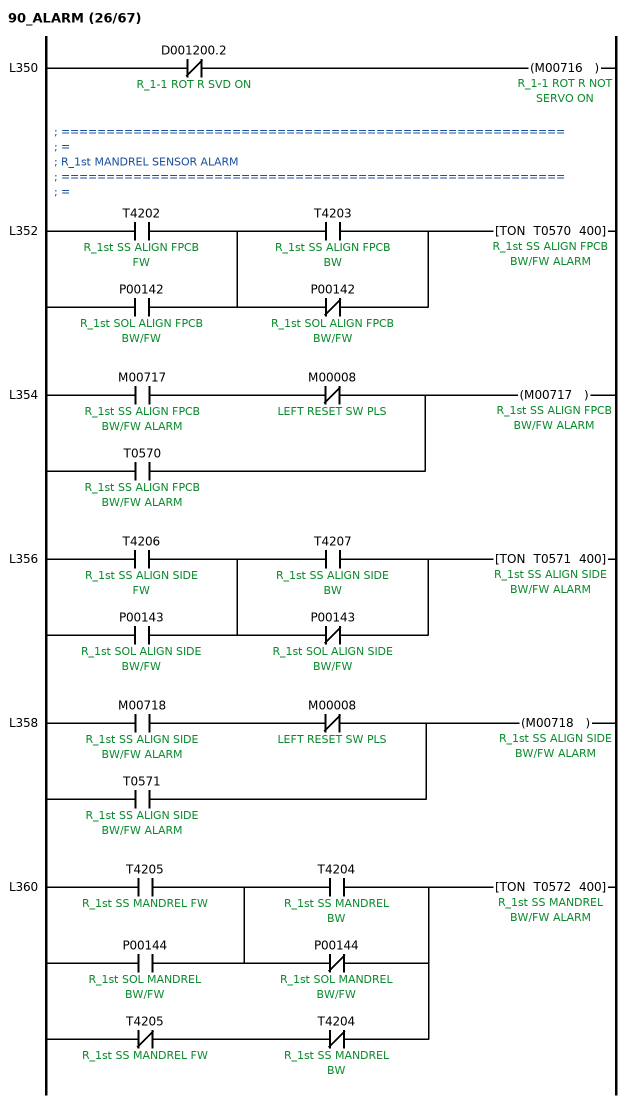
; L350
LOAD NOT  D001200.2	// R_1-1 ROT R SVD ON
OUT       M00716	// R_1-1 ROT R NOT SERVO ON
// =========================================================
// 
//        R_1st MANDREL SENSOR ALARM
// 
// =========================================================
; L352
LOAD      T4202	// R_1st SS ALIGN FPCB FW
OR        P00142	// R_1st SOL ALIGN FPCB BW/FW
LOAD      T4203	// R_1st SS ALIGN FPCB BW
OR NOT    P00142	// R_1st SOL ALIGN FPCB BW/FW
AND LOAD
TON       T0570 400	// R_1st SS ALIGN FPCB BW/FW ALARM
; L354
LOAD      M00717	// R_1st SS ALIGN FPCB BW/FW ALARM
AND NOT   M00008	// LEFT RESET SW PLS
OR        T0570	// R_1st SS ALIGN FPCB BW/FW ALARM
OUT       M00717	// R_1st SS ALIGN FPCB BW/FW ALARM
; L356
LOAD      T4206	// R_1st SS ALIGN SIDE FW
OR        P00143	// R_1st SOL ALIGN SIDE BW/FW
LOAD      T4207	// R_1st SS ALIGN SIDE BW
OR NOT    P00143	// R_1st SOL ALIGN SIDE BW/FW
AND LOAD
TON       T0571 400	// R_1st SS ALIGN SIDE BW/FW ALARM
; L358
LOAD      M00718	// R_1st SS ALIGN SIDE BW/FW ALARM
AND NOT   M00008	// LEFT RESET SW PLS
OR        T0571	// R_1st SS ALIGN SIDE BW/FW ALARM
OUT       M00718	// R_1st SS ALIGN SIDE BW/FW ALARM
; L360
LOAD      T4205	// R_1st SS MANDREL FW
OR        P00144	// R_1st SOL MANDREL BW/FW
LOAD      T4204	// R_1st SS MANDREL BW
OR NOT    P00144	// R_1st SOL MANDREL BW/FW
AND LOAD
LOAD NOT  T4205	// R_1st SS MANDREL FW
AND NOT   T4204	// R_1st SS MANDREL BW
OR LOAD
TON       T0572 400	// R_1st SS MANDREL BW/FW ALARM

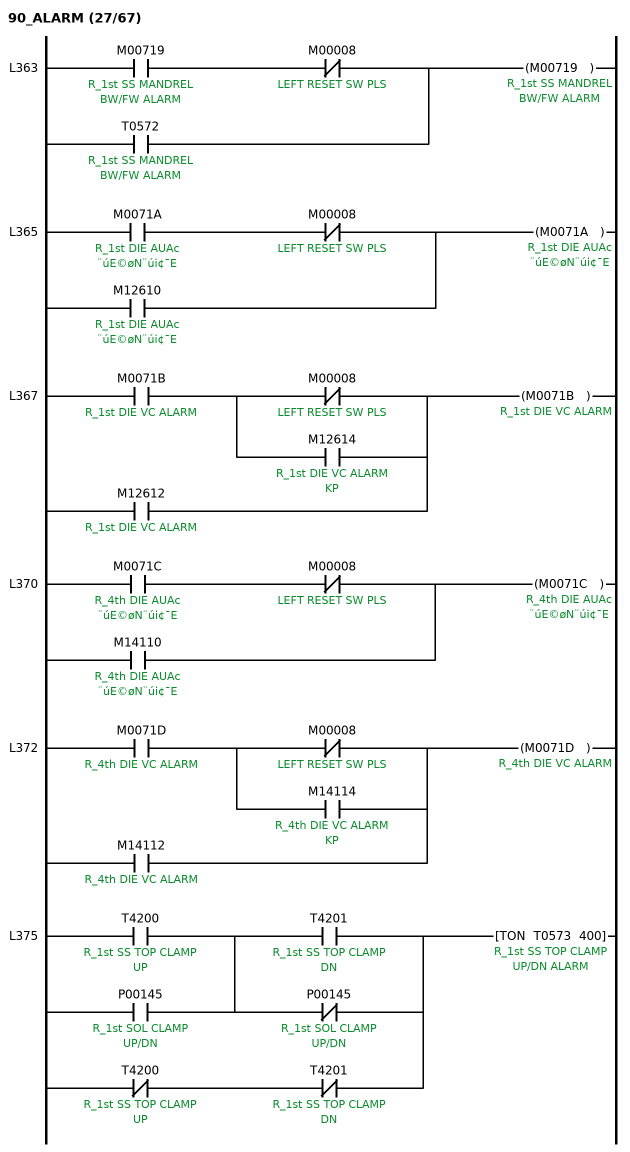
; L363
LOAD      M00719	// R_1st SS MANDREL BW/FW ALARM
AND NOT   M00008	// LEFT RESET SW PLS
OR        T0572	// R_1st SS MANDREL BW/FW ALARM
OUT       M00719	// R_1st SS MANDREL BW/FW ALARM
; L365
LOAD      M0071A	// R_1st DIE AUAc ¨úE©øN¨úi¢¯E
AND NOT   M00008	// LEFT RESET SW PLS
OR        M12610	// R_1st DIE AUAc ¨úE©øN¨úi¢¯E
OUT       M0071A	// R_1st DIE AUAc ¨úE©øN¨úi¢¯E
; L367
LOAD      M0071B	// R_1st DIE VC ALARM
LOAD NOT  M00008	// LEFT RESET SW PLS
OR        M12614	// R_1st DIE VC ALARM KP
AND LOAD
OR        M12612	// R_1st DIE VC ALARM
OUT       M0071B	// R_1st DIE VC ALARM
; L370
LOAD      M0071C	// R_4th DIE AUAc ¨úE©øN¨úi¢¯E
AND NOT   M00008	// LEFT RESET SW PLS
OR        M14110	// R_4th DIE AUAc ¨úE©øN¨úi¢¯E
OUT       M0071C	// R_4th DIE AUAc ¨úE©øN¨úi¢¯E
; L372
LOAD      M0071D	// R_4th DIE VC ALARM
LOAD NOT  M00008	// LEFT RESET SW PLS
OR        M14114	// R_4th DIE VC ALARM KP
AND LOAD
OR        M14112	// R_4th DIE VC ALARM
OUT       M0071D	// R_4th DIE VC ALARM
; L375
LOAD      T4200	// R_1st SS TOP CLAMP UP
OR        P00145	// R_1st SOL CLAMP UP/DN
LOAD      T4201	// R_1st SS TOP CLAMP DN
OR NOT    P00145	// R_1st SOL CLAMP UP/DN
AND LOAD
LOAD NOT  T4200	// R_1st SS TOP CLAMP UP
AND NOT   T4201	// R_1st SS TOP CLAMP DN
OR LOAD
TON       T0573 400	// R_1st SS TOP CLAMP UP/DN ALARM

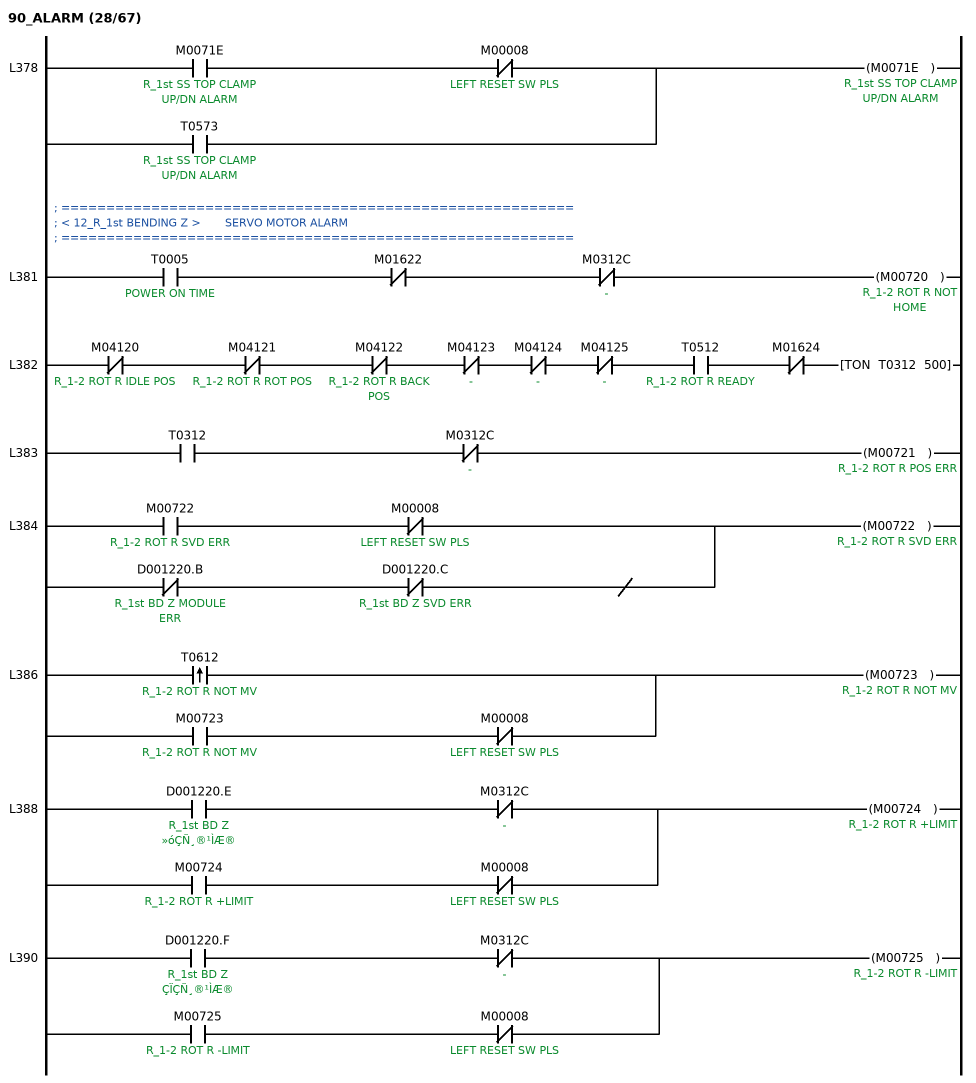
; L378
LOAD      M0071E	// R_1st SS TOP CLAMP UP/DN ALARM
AND NOT   M00008	// LEFT RESET SW PLS
OR        T0573	// R_1st SS TOP CLAMP UP/DN ALARM
OUT       M0071E	// R_1st SS TOP CLAMP UP/DN ALARM
// =========================================================
// 
//        < 12_R_1st BENDING Z >       SERVO MOTOR ALARM
// 
// =========================================================
; L381
LOAD      T0005	// POWER ON TIME
AND NOT   M01622
AND NOT   M0312C	// -
OUT       M00720	// R_1-2 ROT R NOT HOME
; L382
LOAD NOT  M04120	// R_1-2 ROT R IDLE POS
AND NOT   M04121	// R_1-2 ROT R ROT POS
AND NOT   M04122	// R_1-2 ROT R BACK POS
AND NOT   M04123	// -
AND NOT   M04124	// -
AND NOT   M04125	// -
AND       T0512	// R_1-2 ROT R READY
AND NOT   M01624
TON       T0312 500
; L383
LOAD      T0312
AND NOT   M0312C	// -
OUT       M00721	// R_1-2 ROT R POS ERR
; L384
LOAD      M00722	// R_1-2 ROT R SVD ERR
AND NOT   M00008	// LEFT RESET SW PLS
LOAD NOT  D001220.B	// R_1st BD Z MODULE ERR
AND NOT   D001220.C	// R_1st BD Z SVD ERR
NOT
OR LOAD
OUT       M00722	// R_1-2 ROT R SVD ERR
; L386
LOADP     T0612	// R_1-2 ROT R NOT MV
LOAD      M00723	// R_1-2 ROT R NOT MV
AND NOT   M00008	// LEFT RESET SW PLS
OR LOAD
OUT       M00723	// R_1-2 ROT R NOT MV
; L388
LOAD      D001220.E	// R_1st BD Z »óÇÑ¸®¹ÌÆ®
AND NOT   M0312C	// -
LOAD      M00724	// R_1-2 ROT R +LIMIT
AND NOT   M00008	// LEFT RESET SW PLS
OR LOAD
OUT       M00724	// R_1-2 ROT R +LIMIT
; L390
LOAD      D001220.F	// R_1st BD Z ÇÏÇÑ¸®¹ÌÆ®
AND NOT   M0312C	// -
LOAD      M00725	// R_1-2 ROT R -LIMIT
AND NOT   M00008	// LEFT RESET SW PLS
OR LOAD
OUT       M00725	// R_1-2 ROT R -LIMIT

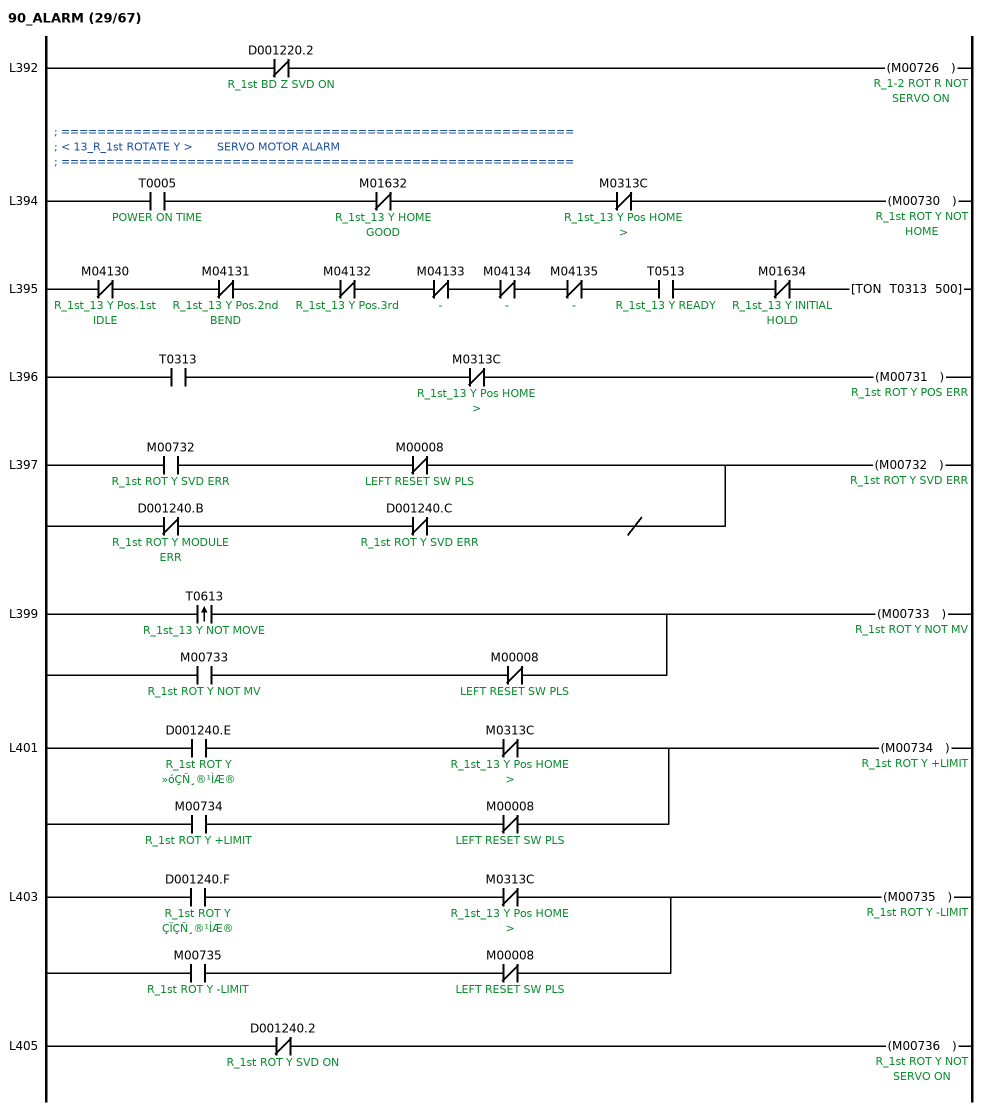
; L392
LOAD NOT  D001220.2	// R_1st BD Z SVD ON
OUT       M00726	// R_1-2 ROT R NOT SERVO ON
// =========================================================
// 
//        < 13_R_1st ROTATE Y >       SERVO MOTOR ALARM
// 
// =========================================================
; L394
LOAD      T0005	// POWER ON TIME
AND NOT   M01632	// R_1st_13 Y HOME GOOD
AND NOT   M0313C	// R_1st_13 Y Pos HOME >
OUT       M00730	// R_1st ROT Y NOT HOME
; L395
LOAD NOT  M04130	// R_1st_13 Y Pos.1st IDLE
AND NOT   M04131	// R_1st_13 Y Pos.2nd BEND
AND NOT   M04132	// R_1st_13 Y Pos.3rd
AND NOT   M04133	// -
AND NOT   M04134	// -
AND NOT   M04135	// -
AND       T0513	// R_1st_13 Y READY
AND NOT   M01634	// R_1st_13 Y INITIAL HOLD
TON       T0313 500
; L396
LOAD      T0313
AND NOT   M0313C	// R_1st_13 Y Pos HOME >
OUT       M00731	// R_1st ROT Y POS ERR
; L397
LOAD      M00732	// R_1st ROT Y SVD ERR
AND NOT   M00008	// LEFT RESET SW PLS
LOAD NOT  D001240.B	// R_1st ROT Y MODULE ERR
AND NOT   D001240.C	// R_1st ROT Y SVD ERR
NOT
OR LOAD
OUT       M00732	// R_1st ROT Y SVD ERR
; L399
LOADP     T0613	// R_1st_13 Y NOT MOVE
LOAD      M00733	// R_1st ROT Y NOT MV
AND NOT   M00008	// LEFT RESET SW PLS
OR LOAD
OUT       M00733	// R_1st ROT Y NOT MV
; L401
LOAD      D001240.E	// R_1st ROT Y »óÇÑ¸®¹ÌÆ®
AND NOT   M0313C	// R_1st_13 Y Pos HOME >
LOAD      M00734	// R_1st ROT Y +LIMIT
AND NOT   M00008	// LEFT RESET SW PLS
OR LOAD
OUT       M00734	// R_1st ROT Y +LIMIT
; L403
LOAD      D001240.F	// R_1st ROT Y ÇÏÇÑ¸®¹ÌÆ®
AND NOT   M0313C	// R_1st_13 Y Pos HOME >
LOAD      M00735	// R_1st ROT Y -LIMIT
AND NOT   M00008	// LEFT RESET SW PLS
OR LOAD
OUT       M00735	// R_1st ROT Y -LIMIT
; L405
LOAD NOT  D001240.2	// R_1st ROT Y SVD ON
OUT       M00736	// R_1st ROT Y NOT SERVO ON

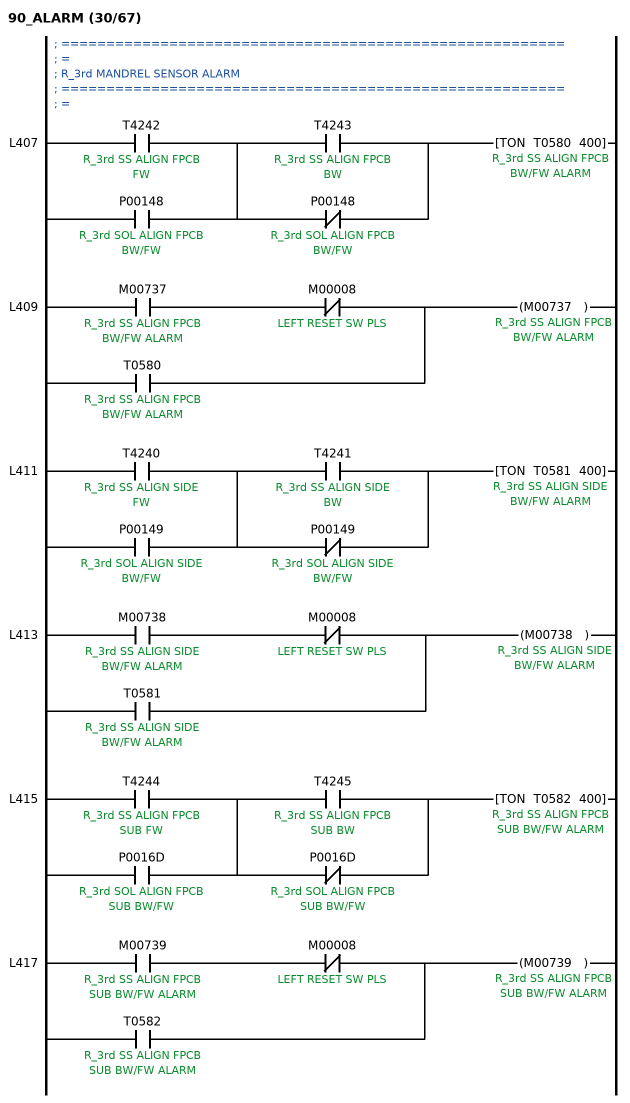
// =========================================================
// 
//        R_3rd MANDREL SENSOR ALARM
// 
// =========================================================
; L407
LOAD      T4242	// R_3rd SS ALIGN FPCB FW
OR        P00148	// R_3rd SOL ALIGN FPCB BW/FW
LOAD      T4243	// R_3rd SS ALIGN FPCB BW
OR NOT    P00148	// R_3rd SOL ALIGN FPCB BW/FW
AND LOAD
TON       T0580 400	// R_3rd SS ALIGN FPCB BW/FW ALARM
; L409
LOAD      M00737	// R_3rd SS ALIGN FPCB BW/FW ALARM
AND NOT   M00008	// LEFT RESET SW PLS
OR        T0580	// R_3rd SS ALIGN FPCB BW/FW ALARM
OUT       M00737	// R_3rd SS ALIGN FPCB BW/FW ALARM
; L411
LOAD      T4240	// R_3rd SS ALIGN SIDE FW
OR        P00149	// R_3rd SOL ALIGN SIDE BW/FW
LOAD      T4241	// R_3rd SS ALIGN SIDE BW
OR NOT    P00149	// R_3rd SOL ALIGN SIDE BW/FW
AND LOAD
TON       T0581 400	// R_3rd SS ALIGN SIDE BW/FW ALARM
; L413
LOAD      M00738	// R_3rd SS ALIGN SIDE BW/FW ALARM
AND NOT   M00008	// LEFT RESET SW PLS
OR        T0581	// R_3rd SS ALIGN SIDE BW/FW ALARM
OUT       M00738	// R_3rd SS ALIGN SIDE BW/FW ALARM
; L415
LOAD      T4244	// R_3rd SS ALIGN FPCB SUB FW
OR        P0016D	// R_3rd SOL ALIGN FPCB SUB BW/FW
LOAD      T4245	// R_3rd SS ALIGN FPCB SUB BW
OR NOT    P0016D	// R_3rd SOL ALIGN FPCB SUB BW/FW
AND LOAD
TON       T0582 400	// R_3rd SS ALIGN FPCB SUB BW/FW ALARM
; L417
LOAD      M00739	// R_3rd SS ALIGN FPCB SUB BW/FW ALARM
AND NOT   M00008	// LEFT RESET SW PLS
OR        T0582	// R_3rd SS ALIGN FPCB SUB BW/FW ALARM
OUT       M00739	// R_3rd SS ALIGN FPCB SUB BW/FW ALARM

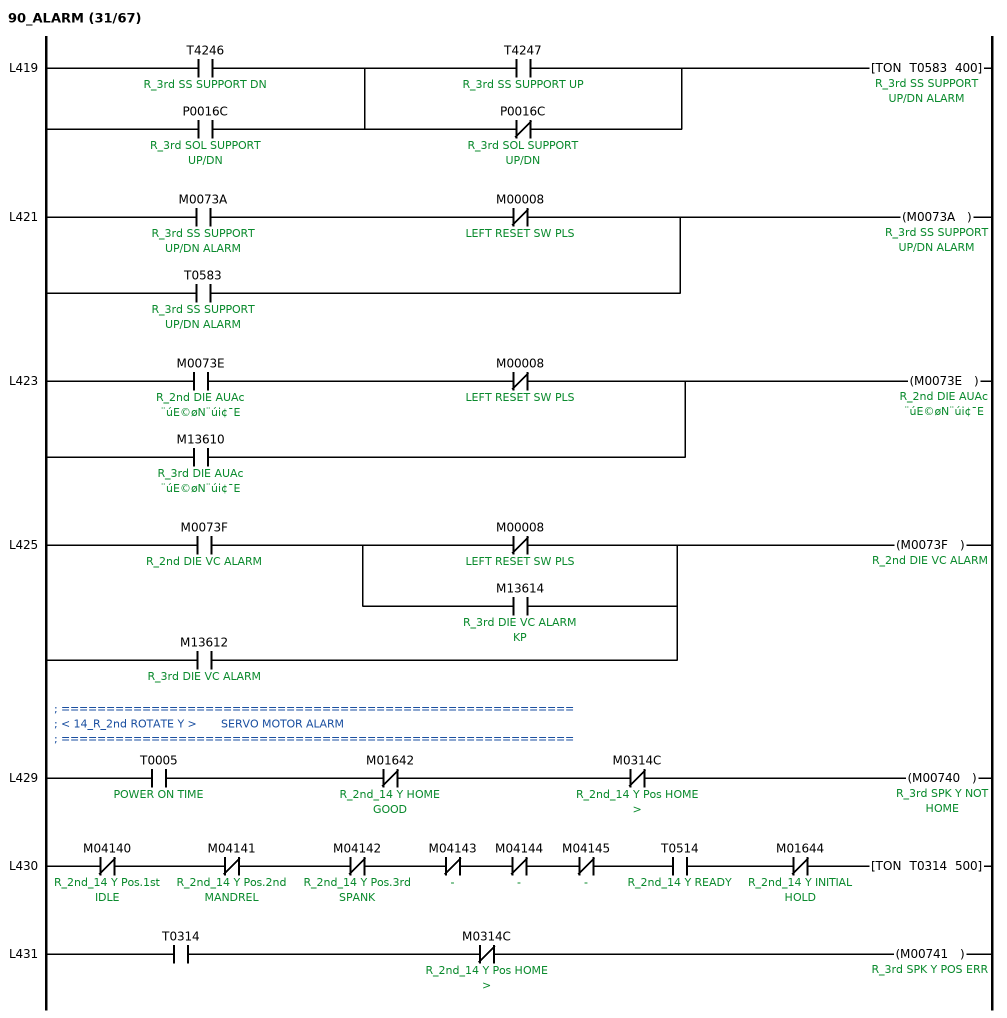
; L419
LOAD      T4246	// R_3rd SS SUPPORT DN
OR        P0016C	// R_3rd SOL SUPPORT UP/DN
LOAD      T4247	// R_3rd SS SUPPORT UP
OR NOT    P0016C	// R_3rd SOL SUPPORT UP/DN
AND LOAD
TON       T0583 400	// R_3rd SS SUPPORT UP/DN ALARM
; L421
LOAD      M0073A	// R_3rd SS SUPPORT UP/DN ALARM
AND NOT   M00008	// LEFT RESET SW PLS
OR        T0583	// R_3rd SS SUPPORT UP/DN ALARM
OUT       M0073A	// R_3rd SS SUPPORT UP/DN ALARM
; L423
LOAD      M0073E	// R_2nd DIE AUAc ¨úE©øN¨úi¢¯E
AND NOT   M00008	// LEFT RESET SW PLS
OR        M13610	// R_3rd DIE AUAc ¨úE©øN¨úi¢¯E
OUT       M0073E	// R_2nd DIE AUAc ¨úE©øN¨úi¢¯E
; L425
LOAD      M0073F	// R_2nd DIE VC ALARM
LOAD NOT  M00008	// LEFT RESET SW PLS
OR        M13614	// R_3rd DIE VC ALARM KP
AND LOAD
OR        M13612	// R_3rd DIE VC ALARM
OUT       M0073F	// R_2nd DIE VC ALARM
// =========================================================
// 
//        < 14_R_2nd ROTATE Y >       SERVO MOTOR ALARM
// 
// =========================================================
; L429
LOAD      T0005	// POWER ON TIME
AND NOT   M01642	// R_2nd_14 Y HOME GOOD
AND NOT   M0314C	// R_2nd_14 Y Pos HOME >
OUT       M00740	// R_3rd SPK Y NOT HOME
; L430
LOAD NOT  M04140	// R_2nd_14 Y Pos.1st IDLE
AND NOT   M04141	// R_2nd_14 Y Pos.2nd MANDREL
AND NOT   M04142	// R_2nd_14 Y Pos.3rd SPANK
AND NOT   M04143	// -
AND NOT   M04144	// -
AND NOT   M04145	// -
AND       T0514	// R_2nd_14 Y READY
AND NOT   M01644	// R_2nd_14 Y INITIAL HOLD
TON       T0314 500
; L431
LOAD      T0314
AND NOT   M0314C	// R_2nd_14 Y Pos HOME >
OUT       M00741	// R_3rd SPK Y POS ERR

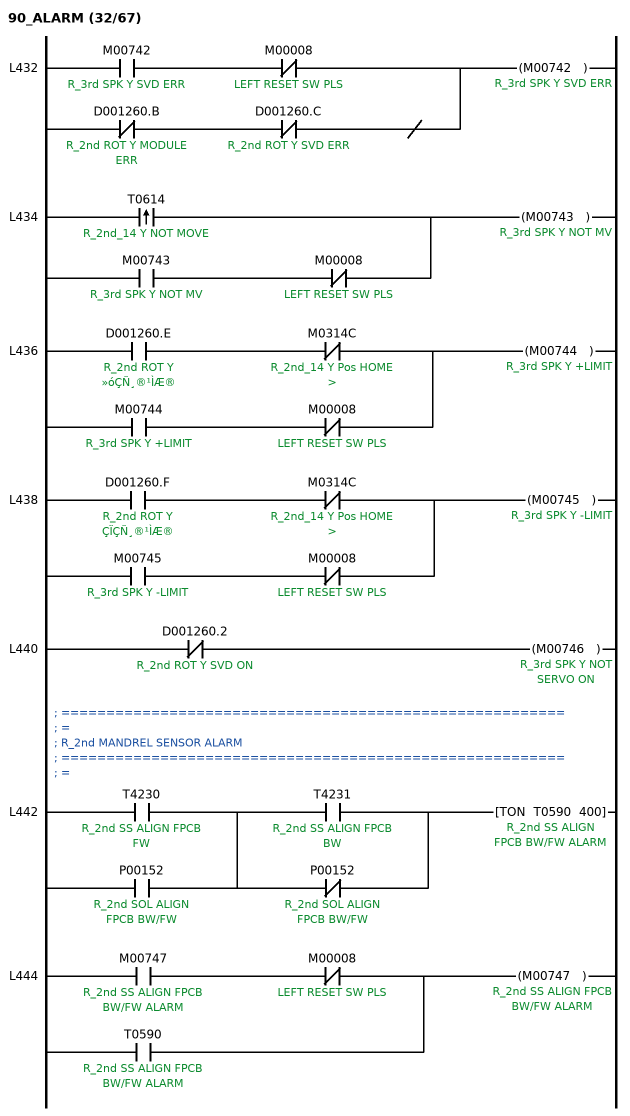
; L432
LOAD      M00742	// R_3rd SPK Y SVD ERR
AND NOT   M00008	// LEFT RESET SW PLS
LOAD NOT  D001260.B	// R_2nd ROT Y MODULE ERR
AND NOT   D001260.C	// R_2nd ROT Y SVD ERR
NOT
OR LOAD
OUT       M00742	// R_3rd SPK Y SVD ERR
; L434
LOADP     T0614	// R_2nd_14 Y NOT MOVE
LOAD      M00743	// R_3rd SPK Y NOT MV
AND NOT   M00008	// LEFT RESET SW PLS
OR LOAD
OUT       M00743	// R_3rd SPK Y NOT MV
; L436
LOAD      D001260.E	// R_2nd ROT Y »óÇÑ¸®¹ÌÆ®
AND NOT   M0314C	// R_2nd_14 Y Pos HOME >
LOAD      M00744	// R_3rd SPK Y +LIMIT
AND NOT   M00008	// LEFT RESET SW PLS
OR LOAD
OUT       M00744	// R_3rd SPK Y +LIMIT
; L438
LOAD      D001260.F	// R_2nd ROT Y ÇÏÇÑ¸®¹ÌÆ®
AND NOT   M0314C	// R_2nd_14 Y Pos HOME >
LOAD      M00745	// R_3rd SPK Y -LIMIT
AND NOT   M00008	// LEFT RESET SW PLS
OR LOAD
OUT       M00745	// R_3rd SPK Y -LIMIT
; L440
LOAD NOT  D001260.2	// R_2nd ROT Y SVD ON
OUT       M00746	// R_3rd SPK Y NOT SERVO ON
// =========================================================
// 
//        R_2nd MANDREL SENSOR ALARM
// 
// =========================================================
; L442
LOAD      T4230	// R_2nd SS ALIGN FPCB FW
OR        P00152	// R_2nd SOL ALIGN FPCB BW/FW
LOAD      T4231	// R_2nd SS ALIGN FPCB BW
OR NOT    P00152	// R_2nd SOL ALIGN FPCB BW/FW
AND LOAD
TON       T0590 400	// R_2nd SS ALIGN FPCB BW/FW ALARM
; L444
LOAD      M00747	// R_2nd SS ALIGN FPCB BW/FW ALARM
AND NOT   M00008	// LEFT RESET SW PLS
OR        T0590	// R_2nd SS ALIGN FPCB BW/FW ALARM
OUT       M00747	// R_2nd SS ALIGN FPCB BW/FW ALARM

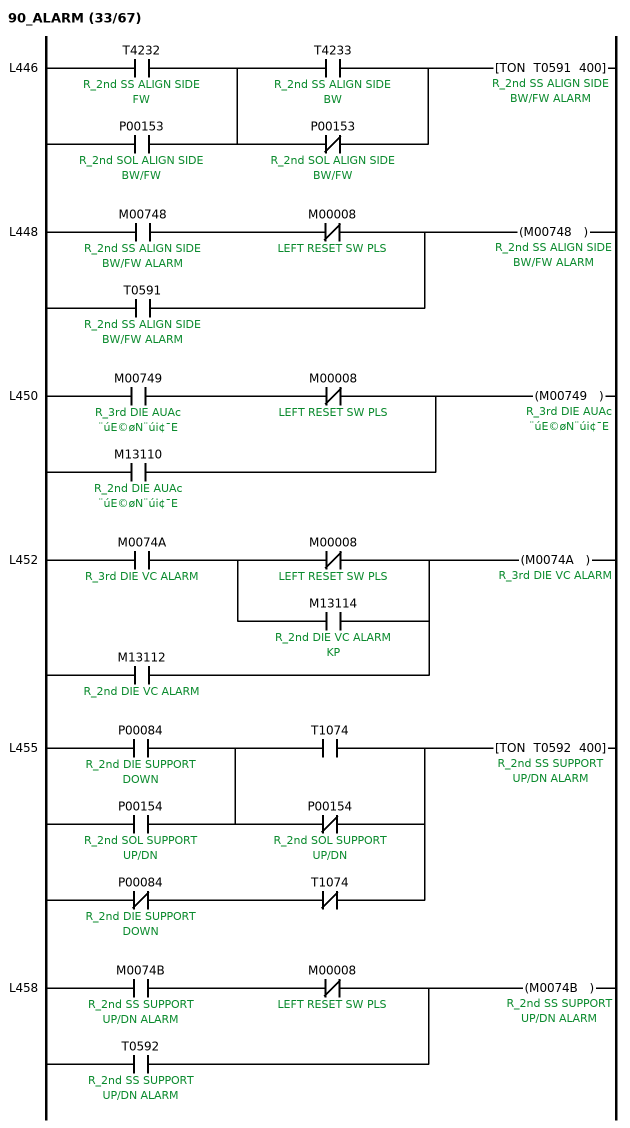
; L446
LOAD      T4232	// R_2nd SS ALIGN SIDE FW
OR        P00153	// R_2nd SOL ALIGN SIDE BW/FW
LOAD      T4233	// R_2nd SS ALIGN SIDE BW
OR NOT    P00153	// R_2nd SOL ALIGN SIDE BW/FW
AND LOAD
TON       T0591 400	// R_2nd SS ALIGN SIDE BW/FW ALARM
; L448
LOAD      M00748	// R_2nd SS ALIGN SIDE BW/FW ALARM
AND NOT   M00008	// LEFT RESET SW PLS
OR        T0591	// R_2nd SS ALIGN SIDE BW/FW ALARM
OUT       M00748	// R_2nd SS ALIGN SIDE BW/FW ALARM
; L450
LOAD      M00749	// R_3rd DIE AUAc ¨úE©øN¨úi¢¯E
AND NOT   M00008	// LEFT RESET SW PLS
OR        M13110	// R_2nd DIE AUAc ¨úE©øN¨úi¢¯E
OUT       M00749	// R_3rd DIE AUAc ¨úE©øN¨úi¢¯E
; L452
LOAD      M0074A	// R_3rd DIE VC ALARM
LOAD NOT  M00008	// LEFT RESET SW PLS
OR        M13114	// R_2nd DIE VC ALARM KP
AND LOAD
OR        M13112	// R_2nd DIE VC ALARM
OUT       M0074A	// R_3rd DIE VC ALARM
; L455
LOAD      P00084	// R_2nd DIE SUPPORT DOWN
OR        P00154	// R_2nd SOL SUPPORT UP/DN
LOAD      T1074
OR NOT    P00154	// R_2nd SOL SUPPORT UP/DN
AND LOAD
LOAD NOT  P00084	// R_2nd DIE SUPPORT DOWN
AND NOT   T1074
OR LOAD
TON       T0592 400	// R_2nd SS SUPPORT UP/DN ALARM
; L458
LOAD      M0074B	// R_2nd SS SUPPORT UP/DN ALARM
AND NOT   M00008	// LEFT RESET SW PLS
OR        T0592	// R_2nd SS SUPPORT UP/DN ALARM
OUT       M0074B	// R_2nd SS SUPPORT UP/DN ALARM

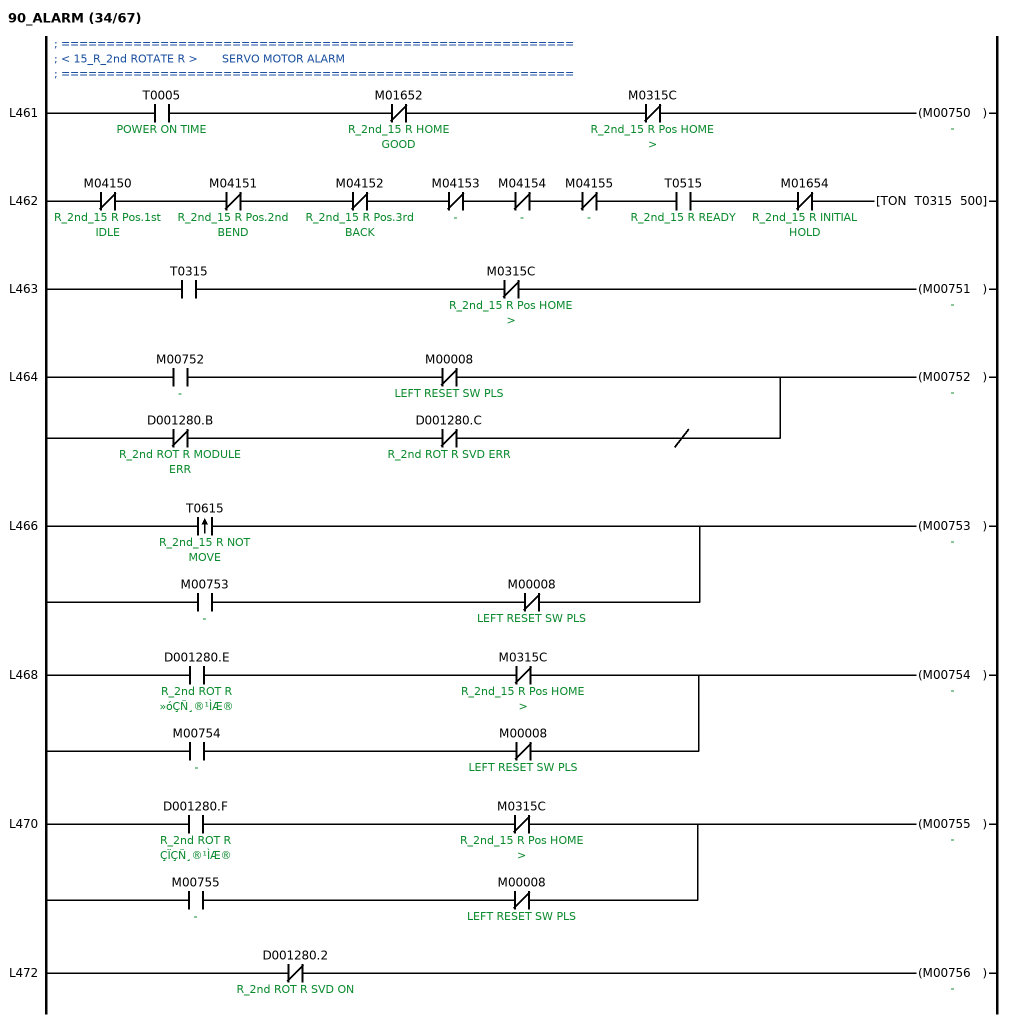
// =========================================================
// 
//        < 15_R_2nd ROTATE R >       SERVO MOTOR ALARM
// 
// =========================================================
; L461
LOAD      T0005	// POWER ON TIME
AND NOT   M01652	// R_2nd_15 R HOME GOOD
AND NOT   M0315C	// R_2nd_15 R Pos HOME >
OUT       M00750	// -
; L462
LOAD NOT  M04150	// R_2nd_15 R Pos.1st IDLE
AND NOT   M04151	// R_2nd_15 R Pos.2nd BEND
AND NOT   M04152	// R_2nd_15 R Pos.3rd BACK
AND NOT   M04153	// -
AND NOT   M04154	// -
AND NOT   M04155	// -
AND       T0515	// R_2nd_15 R READY
AND NOT   M01654	// R_2nd_15 R INITIAL HOLD
TON       T0315 500
; L463
LOAD      T0315
AND NOT   M0315C	// R_2nd_15 R Pos HOME >
OUT       M00751	// -
; L464
LOAD      M00752	// -
AND NOT   M00008	// LEFT RESET SW PLS
LOAD NOT  D001280.B	// R_2nd ROT R MODULE ERR
AND NOT   D001280.C	// R_2nd ROT R SVD ERR
NOT
OR LOAD
OUT       M00752	// -
; L466
LOADP     T0615	// R_2nd_15 R NOT MOVE
LOAD      M00753	// -
AND NOT   M00008	// LEFT RESET SW PLS
OR LOAD
OUT       M00753	// -
; L468
LOAD      D001280.E	// R_2nd ROT R »óÇÑ¸®¹ÌÆ®
AND NOT   M0315C	// R_2nd_15 R Pos HOME >
LOAD      M00754	// -
AND NOT   M00008	// LEFT RESET SW PLS
OR LOAD
OUT       M00754	// -
; L470
LOAD      D001280.F	// R_2nd ROT R ÇÏÇÑ¸®¹ÌÆ®
AND NOT   M0315C	// R_2nd_15 R Pos HOME >
LOAD      M00755	// -
AND NOT   M00008	// LEFT RESET SW PLS
OR LOAD
OUT       M00755	// -
; L472
LOAD NOT  D001280.2	// R_2nd ROT R SVD ON
OUT       M00756	// -

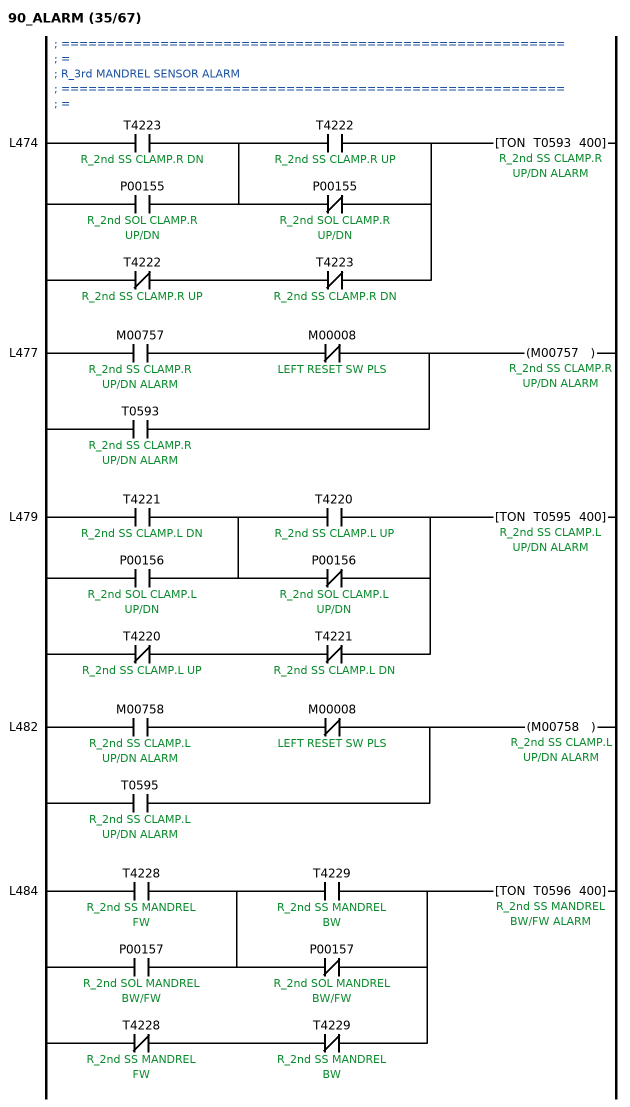
// =========================================================
// 
//        R_3rd MANDREL SENSOR ALARM
// 
// =========================================================
; L474
LOAD      T4223	// R_2nd SS CLAMP.R DN
OR        P00155	// R_2nd SOL CLAMP.R UP/DN
LOAD      T4222	// R_2nd SS CLAMP.R UP
OR NOT    P00155	// R_2nd SOL CLAMP.R UP/DN
AND LOAD
LOAD NOT  T4222	// R_2nd SS CLAMP.R UP
AND NOT   T4223	// R_2nd SS CLAMP.R DN
OR LOAD
TON       T0593 400	// R_2nd SS CLAMP.R UP/DN ALARM
; L477
LOAD      M00757	// R_2nd SS CLAMP.R UP/DN ALARM
AND NOT   M00008	// LEFT RESET SW PLS
OR        T0593	// R_2nd SS CLAMP.R UP/DN ALARM
OUT       M00757	// R_2nd SS CLAMP.R UP/DN ALARM
; L479
LOAD      T4221	// R_2nd SS CLAMP.L DN
OR        P00156	// R_2nd SOL CLAMP.L UP/DN
LOAD      T4220	// R_2nd SS CLAMP.L UP
OR NOT    P00156	// R_2nd SOL CLAMP.L UP/DN
AND LOAD
LOAD NOT  T4220	// R_2nd SS CLAMP.L UP
AND NOT   T4221	// R_2nd SS CLAMP.L DN
OR LOAD
TON       T0595 400	// R_2nd SS CLAMP.L UP/DN ALARM
; L482
LOAD      M00758	// R_2nd SS CLAMP.L UP/DN ALARM
AND NOT   M00008	// LEFT RESET SW PLS
OR        T0595	// R_2nd SS CLAMP.L UP/DN ALARM
OUT       M00758	// R_2nd SS CLAMP.L UP/DN ALARM
; L484
LOAD      T4228	// R_2nd SS MANDREL FW
OR        P00157	// R_2nd SOL MANDREL BW/FW
LOAD      T4229	// R_2nd SS MANDREL BW
OR NOT    P00157	// R_2nd SOL MANDREL BW/FW
AND LOAD
LOAD NOT  T4228	// R_2nd SS MANDREL FW
AND NOT   T4229	// R_2nd SS MANDREL BW
OR LOAD
TON       T0596 400	// R_2nd SS MANDREL BW/FW ALARM

